// TIA Portal V19 program export: 0 tag tables, 0 data types, 49 data blocks, 112 code blocks (in call order from the OBs), 34 instance data blocks

DATA_BLOCK "Analogwerte"   // DB1110
{ S7_Optimized_Access := 'TRUE' }
// stored: AutoNumber false, MemoryReserve 100
   VAR RETAIN
      "LF_CM01.BN01" : Struct   // Leitfähigkeit Bypass Filterpumpe
         MB_min : Real := 0.0;
         MB_max : Real := 2000.0;   // mS
         UG_Alarm : Real := -0.5;
         OG_Alarm : Real := 2200.0;
         GF : Real := 0.5;
         Drahtbruch : Bool := FALSE;
         ungueltig : Bool := FALSE;
      END_STRUCT;
      "LF_CM01.BN02" : Struct   // Leitfähigkeit Düsen Umwälzung
         MB_min : Real := 0.0;
         MB_max : Real := 2000.0;   // mS
         UG_Alarm : Real := -0.5;
         OG_Alarm : Real := 2200.0;
         GF : Real := 0.5;
         Drahtbruch : Bool := FALSE;
         ungueltig : Bool := FALSE;
      END_STRUCT;
      "LF_CM02.BN03" : Struct   // Leitfähigkeit Bypass Filterpumpe
         MB_min : Real := 0.0;
         MB_max : Real := 2000.0;   // mS
         UG_Alarm : Real := -0.5;
         OG_Alarm : Real := 2200.0;
         GF : Real := 0.5;
         Drahtbruch : Bool := FALSE;
         ungueltig : Bool := FALSE;
      END_STRUCT;
      "LF_CM02.BN04" : Struct   // Leitfähigkeit Düsen Umwälzung
         MB_min : Real := 0.0;
         MB_max : Real := 2000.0;   // mS
         UG_Alarm : Real := -0.5;
         OG_Alarm : Real := 2200.0;
         GF : Real := 0.5;
         Drahtbruch : Bool := FALSE;
         ungueltig : Bool := FALSE;
      END_STRUCT;
      "p_HQ01.BP01" : Struct   // Druck Beutelfiltergehäuse
         MB_min : Real := 0.0;
         MB_max : Real := 4.0;   // bar
         UG_Alarm : Real := -0.5;
         OG_Alarm : Real := 4.5;
         GF : Real := 0.5;
         Drahtbruch : Bool := FALSE;
         ungueltig : Bool := FALSE;
      END_STRUCT;
      "p_HQ02.BP02" : Struct   // Druck Beutelfiltergehäuse
         MB_min : Real := 0.0;
         MB_max : Real := 4.0;   // bar
         UG_Alarm : Real := -0.5;
         OG_Alarm : Real := 4.5;
         GF : Real := 0.5;
         Drahtbruch : Bool := FALSE;
         ungueltig : Bool := FALSE;
      END_STRUCT;
      "p_CM01.BP03" : Struct   // Druck Filterpumpe
         MB_min : Real := 0.0;
         MB_max : Real := 4.0;   // bar
         UG_Alarm : Real := -0.5;
         OG_Alarm : Real := 4.5;
         GF : Real := 0.5;
         Drahtbruch : Bool := FALSE;
         ungueltig : Bool := FALSE;
      END_STRUCT;
      "p_CM01.BP04" : Struct   // Druck Umwälzpumpe
         MB_min : Real := 0.0;
         MB_max : Real := 4.0;   // bar
         UG_Alarm : Real := -0.5;
         OG_Alarm : Real := 4.5;
         GF : Real := 0.5;
         Drahtbruch : Bool := FALSE;
         ungueltig : Bool := FALSE;
      END_STRUCT;
      "p_CM03.BP05" : Struct   // Druck Umwäzpumpe
         MB_min : Real := 0.0;
         MB_max : Real := 4.0;   // bar
         UG_Alarm : Real := -0.5;
         OG_Alarm : Real := 4.5;
         GF : Real := 0.5;
         Drahtbruch : Bool := FALSE;
         ungueltig : Bool := FALSE;
      END_STRUCT;
      "p_CM02.BP06" : Struct   // Druck Filterpumpe
         MB_min : Real := 0.0;
         MB_max : Real := 4.0;   // bar
         UG_Alarm : Real := -0.5;
         OG_Alarm : Real := 4.5;
         GF : Real := 0.5;
         Drahtbruch : Bool := FALSE;
         ungueltig : Bool := FALSE;
      END_STRUCT;
      "p_CM02.BP07" : Struct   // Druck Umwälzpumpe
         MB_min : Real := 0.0;
         MB_max : Real := 4.0;   // bar
         UG_Alarm : Real := -0.5;
         OG_Alarm : Real := 4.5;
         GF : Real := 0.5;
         Drahtbruch : Bool := FALSE;
         ungueltig : Bool := FALSE;
      END_STRUCT;
      "p_CM04.BP08" : Struct   // Druck Umwäzpumpe
         MB_min : Real := 0.0;
         MB_max : Real := 4.0;   // bar
         UG_Alarm : Real := -0.5;
         OG_Alarm : Real := 4.5;
         GF : Real := 0.5;
         Drahtbruch : Bool := FALSE;
         ungueltig : Bool := FALSE;
      END_STRUCT;
      "p_CM05.BP09" : Struct   // Druck Pumpe Entleerung Sammeltank
         MB_min : Real := 0.0;
         MB_max : Real := 4.0;   // bar
         UG_Alarm : Real := -0.5;
         OG_Alarm : Real := 4.5;
         GF : Real := 0.5;
         Drahtbruch : Bool := FALSE;
         ungueltig : Bool := FALSE;
      END_STRUCT;
      "Dfl_GP01.BF01" : Struct   // Durchfluss Versorgung Frischsäure
         MB_min : Real := 0.0;
         MB_max : Real := 2000.0;   // ml/s
         UG_Alarm : Real := -0.5;
         OG_Alarm : Real := 2200.0;
         GF : Real := 0.5;
         Drahtbruch : Bool := FALSE;
         ungueltig : Bool := FALSE;
      END_STRUCT;
      "Dfl_GP02.BF02" : Struct   // Durchfluss Entsorgung Altsäure
         MB_min : Real := 0.0;
         MB_max : Real := 2000.0;   // ml/s
         UG_Alarm : Real := -0.5;
         OG_Alarm : Real := 2200.0;
         GF : Real := 0.5;
         Drahtbruch : Bool := FALSE;
         ungueltig : Bool := FALSE;
      END_STRUCT;
      "Niv_GP01.BL30" : Struct   // Füllstand Versorgung Frischsäure
         MB_min : Real := 0.0;
         MB_max : Real := 100.0;   // %
         UG_Alarm : Real := -0.5;
         OG_Alarm : Real := 110.0;
         GF : Real := 0.5;
         Drahtbruch : Bool := FALSE;
         ungueltig : Bool := FALSE;
      END_STRUCT;
      "Niv_GP02.BL31" : Struct   // Füllstand Entsorgung Altsäure
         MB_min : Real := 0.0;
         MB_max : Real := 100.0;   // %
         UG_Alarm : Real := -0.5;
         OG_Alarm : Real := 110.0;
         GF : Real := 0.5;
         Drahtbruch : Bool := FALSE;
         ungueltig : Bool := FALSE;
      END_STRUCT;
      pH_WR01 : Struct   // pH-Wert Be-/Entladen
         MB_min : Real := 0.0;
         MB_max : Real := 100.0;   // %
         UG_Alarm : Real := -0.5;
         OG_Alarm : Real := 110.0;
         GF : Real := 0.5;
         Drahtbruch : Bool := FALSE;
         ungueltig : Bool := FALSE;
      END_STRUCT;
      WZ_1_1 : Struct   // Wägezelle WR04.BW01
         MB_min : Real := 0.0;
         MB_max : Real := 100.0;   // %
         UG_Alarm : Real := -0.5;
         OG_Alarm : Real := 110.0;
         GF : Real := 0.5;
         Drahtbruch : Bool := FALSE;
         ungueltig : Bool := FALSE;
      END_STRUCT;
      WZ_1_2 : Struct   // Wägezelle WR04.BW02
         MB_min : Real := 0.0;
         MB_max : Real := 100.0;   // %
         UG_Alarm : Real := -0.5;
         OG_Alarm : Real := 110.0;
         GF : Real := 0.5;
         Drahtbruch : Bool := FALSE;
         ungueltig : Bool := FALSE;
      END_STRUCT;
      WZ_1_3 : Struct   // Wägezelle WR04.BW03
         MB_min : Real := 0.0;
         MB_max : Real := 100.0;   // %
         UG_Alarm : Real := -0.5;
         OG_Alarm : Real := 110.0;
         GF : Real := 0.5;
         Drahtbruch : Bool := FALSE;
         ungueltig : Bool := FALSE;
      END_STRUCT;
      WZ_1_4 : Struct   // Wägezelle WR04.BW04
         MB_min : Real := 0.0;
         MB_max : Real := 100.0;   // %
         UG_Alarm : Real := -0.5;
         OG_Alarm : Real := 110.0;
         GF : Real := 0.5;
         Drahtbruch : Bool := FALSE;
         ungueltig : Bool := FALSE;
      END_STRUCT;
      WZ_2_1 : Struct   // Wägezelle WR05.BW01
         MB_min : Real := 0.0;
         MB_max : Real := 100.0;   // %
         UG_Alarm : Real := -0.5;
         OG_Alarm : Real := 110.0;
         GF : Real := 0.5;
         Drahtbruch : Bool := FALSE;
         ungueltig : Bool := FALSE;
      END_STRUCT;
      WZ_2_2 : Struct   // Wägezelle WR05.BW01
         MB_min : Real := 0.0;
         MB_max : Real := 100.0;   // %
         UG_Alarm : Real := -0.5;
         OG_Alarm : Real := 110.0;
         GF : Real := 0.5;
         Drahtbruch : Bool := FALSE;
         ungueltig : Bool := FALSE;
      END_STRUCT;
      WZ_2_3 : Struct   // Wägezelle WR05.BW01
         MB_min : Real := 0.0;
         MB_max : Real := 100.0;   // %
         UG_Alarm : Real := -0.5;
         OG_Alarm : Real := 110.0;
         GF : Real := 0.5;
         Drahtbruch : Bool := FALSE;
         ungueltig : Bool := FALSE;
      END_STRUCT;
      WZ_2_4 : Struct   // Wägezelle WR05.BW01
         MB_min : Real := 0.0;
         MB_max : Real := 100.0;   // %
         UG_Alarm : Real := -0.5;
         OG_Alarm : Real := 110.0;
         GF : Real := 0.5;
         Drahtbruch : Bool := FALSE;
         ungueltig : Bool := FALSE;
      END_STRUCT;
      Last_1 : Struct   // Novamat WR04.BW34
         MB_min : Real := 0.0;
         MB_max : Real := 100.0;   // %
         UG_Alarm : Real := -0.5;
         OG_Alarm : Real := 110.0;
         GF : Real := 0.5;
         Drahtbruch : Bool := FALSE;
         ungueltig : Bool := FALSE;
      END_STRUCT;
      Last_2 : Struct   // Novamat WR05.BW43
         MB_min : Real := 0.0;
         MB_max : Real := 100.0;   // %
         UG_Alarm : Real := -0.5;
         OG_Alarm : Real := 110.0;
         GF : Real := 0.5;
         Drahtbruch : Bool := FALSE;
         ungueltig : Bool := FALSE;
      END_STRUCT;
   END_VAR
BEGIN
END_DATA_BLOCK

DATA_BLOCK "DB_ANLAGE"   // DB1
{ S7_Optimized_Access := 'FALSE' }
AUTHOR : MS
// stored: AutoNumber false
   VAR RETAIN
      BA : Struct   // Betriebsarten
         Not_Aus : Bool := FALSE;   // Not-Aus ist betätigt
         free0 : Bool := FALSE;   // sonst Anlage vom PC bedienen, nur bei BA-Schalter auf Auto
         free1 : Bool := FALSE;   // sonst Automatikbetrieb ist nicht freigegeben
         Tippbetrieb : Bool := FALSE;   // Tippbetrieb
         Handbetrieb : Bool := FALSE;   // Handbetrieb
         Automat_ein : Bool := FALSE;   // Automatikbetrieb möglich
         Automat_aus : Bool := FALSE;   // Automatikbetrieb nicht möglich
         Anlauf_Auto : Bool := FALSE;   // Anlauf Automatik für Scanvorgang WT-Positionen auf letzte Automatikposition
         Einfahr_Stop : Bool := FALSE;   // Stoppt die Einfahrt von WT in die Anlage(Feierabendprogramm)
         Mess_on : Bool := FALSE;   // Einmessung aktiv
         Taktwechsel : Bool := FALSE;   // Taktwechsel durchführen
         SIM_HISPEED : Bool := FALSE;   // * Simulation erfolgt mit doppelter Geschwindigkeit
         Simulation : Bool := FALSE;   // * Simulation eingeschaltet
         COM_RST : Bool := TRUE;   // Complete Restart
         FP_Automat_ein : Bool := FALSE;   // Flankenmerker positive Flanke Taste Automat ein
         newConfig : Bool := FALSE;   // neue Konfiguration (Daten neu verteilen)
      END_STRUCT;
      config : Struct   // Anlagenkonfiguration
         ANZ_FW : Int := 1;   // * Anzahl der Transportwagen in der Anlage
         ANZ_QT : Int := 0;   // * Anzahl der Quertransporte in der Anlage
         ANZ_Reihen : Int := 1;   // * Anzahl der Reihen in der Anlage
         ANZ_Pos : Int := 30;   // * Anzahl der Positionen
         ANZ_WT : Int := 12;   // * Anzahl der vorhandenen WT-Datenbausteine
         ANZ_POS_per_Cyc : Int := 6;   // * Anzahl der bearbeiteten Positionen pro Zyklus
         maxWT_loop : Int := 5;   // * im freien System Anzahl der Befehle der größten Technologieschleife
         Anz_Opt_Pos : Int := 0;   // * Anzahl der in die Optimierungsrechnung eingehenden Positionen
         Anz_GR : Int := 0;   // * Anzahl der Gleichrichter
         Anz_TR : Int := 0;   // * Anzahl der Temperaturregler
         Anz_DZ : Int := 2;   // * Anzahl der Dosierzähler
         Anz_DP : Int := 8;   // * Anzahl Dosierpumpen
         AnaEventInt : Int := 600;   // * Analogevent Intervall
         Taktzeit_typ : Int := 480;   // * typische Taktzeit für Expoberechnung in getakteten Positionen
         Transzeit_typ : Int := 60;   // * typische Zeit für einen Austauschvorgang
         Reihen_Cnfg : Struct
            EndePos_R1 : Int := 30;   // * Reihendefinition, letzte Position in Reihe 1 (immer niedriger als EndePos_R2)
            EndePos_R2 : Int := 0;   // * Reihendefinition, letzte Position in Reihe 2 (immer niedriger als EndePos_R3)
            EndePos_R3 : Int := 0;   // * Reihendefinition, letzte Position in Reihe 3 (immer niedriger als EndePos_R4)
            EndePos_R4 : Int := 0;   // * Reihendefinition, letzte Position in Reihe 4 (immer niedriger als EndePos_R5)
            EndePos_R5 : Int := 0;   // * Reihendefinition, letzte Position in Reihe 5
         END_STRUCT;
         akt_FW : Int := 0;
         Old_Hour_Event : Int := 0;
         PC_exist : Bool := 0;   // * PC-Daten schreiben (es existiert ein EventAbnehmer [FC7])
         Diag_exist : Bool := 0;   // * Diagrammdaten schreiben (Diagrammdaten werden am PC aufgezeichnet)
         Anl_getaktet : Bool := TRUE;   // * 0=Anlage fährt Auftragsorientiert 1=Anlage wird mit Ketten gesteuert
         HW_exist : Bool := TRUE;   // * Höhenwechsel in der Anlage vorhanden
         Pos_absolut : Bool := TRUE;   // * Positionsbestimmung absolut für OB100-Init-Pos (wirkt nicht mehr am FW)
         Opti_exist : Bool := FALSE;   // * Optimierung vorhanden
         AL_Einfahrt : Bool := FALSE;   // Ware aufgeben!!
         Al_Ausfahrt : Bool := FALSE;   // Beladestand räumen!!
         Weg_Zeit_aus : Bool := FALSE;   // * Weg-Zeit-Events nicht schreiben
         EntmFromOpt : Bool := FALSE;   // * Entmetallisierungs-WT werden von der Optimierung berechnet
         M_Q_Hupe : Bool := TRUE;
         HW_Auto_search : Bool := FALSE;   // * FW sucht automatisch nach einer möglichen Höhenwechselposition
         FP_Taste_Reset : Bool := FALSE;
         Time_from_PC : Bool := 0;   // * Zeit wird vom PC gestellt (keine autom. Sommerzeit)
         FP_Stop_Taktende : Bool := FALSE;   // Flankenmerker Stop bei Taktende erreicht
         Temp_MW_aktiv : Bool := 0;   // * Event mittlere Temperatur (Event 18) aktiv
         FP_Einrichten : Bool := FALSE;
         FP_Hand : Bool := TRUE;
         FP_Automatik : Bool := FALSE;
         FP_In_Quitt : Bool := FALSE;   // Flankenmerker Fehlerquittung
         Hub_absolut : Bool := FALSE;   // Hubsesorik Absolutgeber
         Battf : Bool := FALSE;   // Batteriefehler OB81 (Durch Hardwareschalter an SPS "BATT_INDIC") quittierbar
         RESET_STATUS : Bool := FALSE;   // Wiederanlaufmerker nach Reset
         WT_Typ_Afg : Bool := FALSE;   // * WT-Typ wird bei Aufgabe vergeben
         TypChckDetail : Bool := TRUE;   // * WT-Typ wird ohne Maske B#16#F0 geprüft
         QT_Trocken_chk : Bool := FALSE;   // * einschalten, wenn Prüfung auf bit "immer schnell"
         FB9_Takt : Bool := FALSE;   // * FB9 aufrufen obwohl Anlage getaktet
         Use_FB_Ana : Bool := 0;   // * 1=FB110 verwenden 0=klassische Analogwerterfassung FC110
         Check_Profibus : Bool := TRUE;   // * Profibusteilnehmer überwachen! OB86,OB100,DB203,FC203
         NormalB : Bool := FALSE;   // 0: 151 / 161 1: nur 151
         res6 : Bool := FALSE;
         ReqUmsTakt : Bool := FALSE;   // Anforderung Umschaltung auf getaktet
      END_STRUCT;
      IN : Struct   // Hardwareeingänge Anlage
         S_Not_Aus : Bool := FALSE;   // Not-Aus ok
         S_St_Spng : Bool := TRUE;   // Steuerspannung ein
         Quitt_Err : Bool := FALSE;   // Fehlerquittung
         Quitt_Hupe : Bool := FALSE;   // Hupenquittierung
         Reset : Bool := FALSE;   // Reset Anlagenschalter
         Reparatur : Bool := FALSE;   // Reparaturbetrieb
         Lamp_Test : Bool := FALSE;   // Lampentest
         BA_Tipp : Bool := FALSE;   // BA Umschalter Tipp
         BA_Hand : Bool := TRUE;   // BA Umschalter Hand
         BA_Auto : Bool := FALSE;   // BA Umschalter Auto
         Stop_Anlage : Bool := FALSE;   // Anlage hält am Takt- bzw. Schichtende an
         Automat_aus : Bool := FALSE;   // Taste Automatikbetrieb verbieten
         Automat_ein : Bool := FALSE;   // Taste Automatikbetrieb erlauben
         Quit_Err_Galva : Bool := FALSE;   // Fehlerquittung per Galva
         res4 : Bool := FALSE;
         UT_Req : Bool := FALSE;   // Anforderung Umlufttrockner
         ReqEventTakt : Bool := FALSE;   // Anforderung EventTakt
         GR_ok : Bool := FALSE;   // Rückmeldung Event erfolgt
         TR_ok : Bool := FALSE;   // Rückmeldung Event erfolgt
         pH_LF_ok : Bool := TRUE;   // Rückmeldung Event erfolgt
         DP_ok : Bool := FALSE;   // Rückmeldung Event erfolgt
         res11 : Bool := FALSE;
         res12 : Bool := FALSE;
         res13 : Bool := FALSE;
         PC_offline : Bool := FALSE;   // PC-Komunikation ist unterbrochen
         AMS_Restart : Bool := FALSE;   // alle anstehenden Fehler neu senden
         Watch_Profibus : Bool := FALSE;   // Profibusüberwachung eingeschaltet
         res17 : Bool := FALSE;
         res18 : Bool := FALSE;
         res19 : Bool := FALSE;
         res20 : Bool := FALSE;
         AMS_Reset : Bool := FALSE;   // AMS-Reset durchführen (Resetknopf während nicht Tipp)
      END_STRUCT;
      OUT : Struct   // Hardwareausgänge Anlage
         Stoerung_Opt : Bool := FALSE;
         Stoerung_Aku : Bool := FALSE;
         MD_Auto : Bool := FALSE;
         Fehler_Quitt : Bool := FALSE;
         res1 : Bool := FALSE;
         res2 : Bool := FALSE;
         res3 : Bool := FALSE;
         FW_QT_Auto : Bool := FALSE;   // mind. ein FW/QT hat seinen Automatikbefehl noch nicht beendet
         TW_abgelehnt : Bool := FALSE;   // Taktwechsel wurde abgelehnt (durch Fehlerquittung löschen)
         WT_in_Anlage : Bool := FALSE;
         res7 : Bool := FALSE;
         res8 : Bool := FALSE;
         res9 : Bool := FALSE;
         res10 : Bool := FALSE;
         res11 : Bool := FALSE;
         res12 : Bool := FALSE;
         res13 : Bool := FALSE;
         res14 : Bool := FALSE;
         res15 : Bool := FALSE;
         res16 : Bool := FALSE;
         res17 : Bool := FALSE;
         res18 : Bool := FALSE;
         res19 : Bool := FALSE;
         res20 : Bool := FALSE;
         AnzUT_Req : Byte := 16#00;   // Anzahl der UT Anforderungen
      END_STRUCT;
      config2 : Struct
         Anzahl_HW : Int := 1;   // * Anzahl Höhenwechsel (Definition im DB53)
         Woscha_DB_1 : Int := 8;   // Datenbaustein für Wochenschaltuhr 1
         Woscha_DB_2 : Int := 0;   // Datenbaustein für Wochenschaltuhr 2
         Woscha_DB_3 : Int := 0;   // Datenbaustein für Wochenschaltuhr 3
         Woscha_DB_4 : Int := 0;   // Datenbaustein für Wochenschaltuhr 4
         resW4 : Int := 0;
         Anlagentakte : Int := 3;   // Anzahl Takte, welche WT durch die Anlage läuft
         resW6 : Int := 0;
         resW7 : Int := 0;
         resW8 : Int := 0;
         resW9 : Int := 0;
         resW10 : Int := 0;
         resW11 : Int := 0;
         resW12 : Int := 0;
         resW13 : Int := 0;
         resW14 : Int := 0;
         resW15 : Int := 0;
         resW16 : Int := 0;
         resW17 : Int := 0;
         resW18 : Int := 0;
         resW19 : Int := 0;
      END_STRUCT;
      FW1 : Struct
         FW_min : Int := 1;   // * FW Bereich min
         FW_max : Int := 30;   // * FW Bereich max
         RefPos : Int := 0;   // * Referenzposition (bei Absolutpositionierung 0)
         T_Nr : Int := 10;   // * Timer1
         resW : Int := 0;
      END_STRUCT;
      FW2 : Struct
         FW_min : Int := 0;   // * FW Bereich min
         FW_max : Int := 0;   // * FW Bereich max
         RefPos : Int := 0;   // * Referenzposition (bei Absolutpositionierung 0)
         T_Nr : Int := 0;   // * Timer1
         resW : Int := 0;
      END_STRUCT;
      FW3 : Struct
         FW_min : Int := 0;   // * FW Bereich min
         FW_max : Int := 0;   // * FW Bereich max
         RefPos : Int := 0;   // * Referenzposition (bei Absolutpositionierung 0)
         T_Nr : Int := 0;   // * Timer1
         resW : Int := 0;
      END_STRUCT;
      FW4 : Struct
         FW_min : Int := 0;   // * FW Bereich min
         FW_max : Int := 0;   // * FW Bereich max
         RefPos : Int := 0;   // * Referenzposition (bei Absolutpositionierung 0)
         T_Nr : Int := 0;   // * Timer1
         resW : Int := 0;
      END_STRUCT;
      FW5 : Struct
         FW_min : Int := 0;   // * FW Bereich min
         FW_max : Int := 0;   // * FW Bereich max
         RefPos : Int := 0;   // * Referenzposition (bei Absolutpositionierung 0)
         T_Nr : Int := 0;   // * Timer1
         resW : Int := 0;
      END_STRUCT;
      FW6 : Struct
         FW_min : Int := 0;   // * FW Bereich min
         FW_max : Int := 0;   // * FW Bereich max
         RefPos : Int := 0;   // * Referenzposition (bei Absolutpositionierung 0)
         T_Nr : Int := 0;   // * Timer1
         resW : Int := 0;
      END_STRUCT;
      FW7 : Struct
         FW_min : Int := 0;   // * FW Bereich min
         FW_max : Int := 0;   // * FW Bereich max
         RefPos : Int := 0;   // * Referenzposition (bei Absolutpositionierung 0)
         T_Nr : Int := 0;   // * Timer1
         resW : Int := 0;
      END_STRUCT;
      FW8 : Struct
         FW_min : Int := 0;   // * FW Bereich min
         FW_max : Int := 0;   // * FW Bereich max
         RefPos : Int := 0;   // * Referenzposition (bei Absolutpositionierung 0)
         T_Nr : Int := 0;   // * Timer1
         resW : Int := 0;
      END_STRUCT;
      FW9 : Struct
         FW_min : Int := 0;   // * FW Bereich min
         FW_max : Int := 0;   // * FW Bereich max
         RefPos : Int := 0;   // * Referenzposition (bei Absolutpositionierung 0)
         T_Nr : Int := 0;   // * Timer1
         resW : Int := 0;
      END_STRUCT;
      FW10 : Struct
         FW_min : Int := 0;   // * FW Bereich min
         FW_max : Int := 0;   // * FW Bereich max
         RefPos : Int := 0;   // * Referenzposition (bei Absolutpositionierung 0)
         T_Nr : Int := 0;   // * Timer1
         resW : Int := 0;
      END_STRUCT;
      FW11 : Struct
         FW_min : Int := 0;   // * FW Bereich min
         FW_max : Int := 0;   // * FW Bereich max
         RefPos : Int := 0;   // * Referenzposition (bei Absolutpositionierung 0)
         T_Nr : Int := 0;   // * Timer1
         resW : Int := 0;
      END_STRUCT;
      FW12 : Struct
         FW_min : Int := 0;   // * FW Bereich min
         FW_max : Int := 0;   // * FW Bereich max
         RefPos : Int := 0;   // * Referenzposition (bei Absolutpositionierung 0)
         T_Nr : Int := 0;   // * Timer1
         resW : Int := 0;
      END_STRUCT;
      FW13 : Struct
         FW_min : Int := 0;   // * FW Bereich min
         FW_max : Int := 0;   // * FW Bereich max
         RefPos : Int := 0;   // * Referenzposition (bei Absolutpositionierung 0)
         T_Nr : Int := 0;   // * Timer1
         resW : Int := 0;
      END_STRUCT;
      FW14 : Struct
         FW_min : Int := 0;   // * FW Bereich min
         FW_max : Int := 0;   // * FW Bereich max
         RefPos : Int := 0;   // * Referenzposition (bei Absolutpositionierung 0)
         T_Nr : Int := 0;   // * Timer1
         resW : Int := 0;
      END_STRUCT;
      FW15 : Struct
         FW_min : Int := 0;   // * FW Bereich min
         FW_max : Int := 0;   // * FW Bereich max
         RefPos : Int := 0;   // * Referenzposition (bei Absolutpositionierung 0)
         T_Nr : Int := 0;   // * Timer1
         resW : Int := 0;
      END_STRUCT;
      QT1 : Struct
         PosR1 : Byte := 16#00;   // * QT-Reihe1: Positionsnummer der ersten QT-Pos (bei Rückwärtsfahrt letzte Pos)
         PosR2 : Byte := 16#00;   // * QT-Reihe2: Positionsnummer der zweiten QT-Pos
         PosR3 : Byte := 16#00;   // * QT-Reihe3: Positionsnummer der dritten QT-Pos
         PosR4 : Byte := 16#00;   // * QT-Reihe4: Positionsnummer der vierten QT-Pos
         PosR5 : Byte := 16#00;   // * QT-Reihe5: Positionsnummer der fünften QT-Pos
         RefReihe : Byte := 16#00;   // * Referenzreihe nur angeben wenn mitfahrende Sensoren!!
         T_Nr : Int := 0;   // * Timer1
         Ketten_DB : Int := 0;   // * Eintrag == 0 --> QT besitzt keine Kette
      END_STRUCT;
      QT2 : Struct
         PosR1 : Byte := 16#00;   // * QT-Reihe1: Positionsnummer der ersten QT-Pos (bei Rückwärtsfahrt letzte Pos)
         PosR2 : Byte := 16#00;   // * QT-Reihe2: Positionsnummer der zweiten QT-Pos
         PosR3 : Byte := 16#00;   // * QT-Reihe3: Positionsnummer der dritten QT-Pos
         PosR4 : Byte := 16#00;   // * QT-Reihe4: Positionsnummer der vierten QT-Pos
         PosR5 : Byte := 16#00;   // * QT-Reihe5: Positionsnummer der fünften QT-Pos
         RefReihe : Byte := 16#00;   // * Referenzreihe nur angeben wenn mitfahrende Sensoren!!
         T_Nr : Int := 0;   // * Timer1
         Ketten_DB : Int := 0;   // * Eintrag == 0 --> QT besitzt keine Kette
      END_STRUCT;
      QT3 : Struct
         PosR1 : Byte := 16#00;   // * QT-Reihe1: Positionsnummer der ersten QT-Pos (bei Rückwärtsfahrt letzte Pos)
         PosR2 : Byte := 16#00;   // * QT-Reihe2: Positionsnummer der zweiten QT-Pos
         PosR3 : Byte := 16#00;   // * QT-Reihe3: Positionsnummer der dritten QT-Pos
         PosR4 : Byte := 16#00;   // * QT-Reihe4: Positionsnummer der vierten QT-Pos
         PosR5 : Byte := 16#00;   // * QT-Reihe5: Positionsnummer der fünften QT-Pos
         RefReihe : Byte := 16#00;   // * Referenzreihe nur angeben wenn mitfahrende Sensoren!!
         T_Nr : Int := 0;   // * Timer1
         Ketten_DB : Int := 0;   // * Eintrag == 0 --> QT besitzt keine Kette
      END_STRUCT;
      QT4 : Struct
         PosR1 : Byte := 16#00;   // * QT-Reihe1: Positionsnummer der ersten QT-Pos (bei Rückwärtsfahrt letzte Pos)
         PosR2 : Byte := 16#00;   // * QT-Reihe2: Positionsnummer der zweiten QT-Pos
         PosR3 : Byte := 16#00;   // * QT-Reihe3: Positionsnummer der dritten QT-Pos
         PosR4 : Byte := 16#00;   // * QT-Reihe4: Positionsnummer der vierten QT-Pos
         PosR5 : Byte := 16#00;   // * QT-Reihe5: Positionsnummer der fünften QT-Pos
         RefReihe : Byte := 16#00;   // * Referenzreihe nur angeben wenn mitfahrende Sensoren!!
         T_Nr : Int := 0;   // * Timer1
         Ketten_DB : Int := 0;   // * Eintrag == 0 --> QT besitzt keine Kette
      END_STRUCT;
      QT5 : Struct
         PosR1 : Byte := 16#00;   // * QT-Reihe1: Positionsnummer der ersten QT-Pos (bei Rückwärtsfahrt letzte Pos)
         PosR2 : Byte := 16#00;   // * QT-Reihe2: Positionsnummer der zweiten QT-Pos
         PosR3 : Byte := 16#00;   // * QT-Reihe3: Positionsnummer der dritten QT-Pos
         PosR4 : Byte := 16#00;   // * QT-Reihe4: Positionsnummer der vierten QT-Pos
         PosR5 : Byte := 16#00;   // * QT-Reihe5: Positionsnummer der fünften QT-Pos
         RefReihe : Byte := 16#00;   // * Referenzreihe nur angeben wenn mitfahrende Sensoren!!
         T_Nr : Int := 0;   // * Timer1
         Ketten_DB : Int := 0;   // * Eintrag == 0 --> QT besitzt keine Kette
      END_STRUCT;
   END_VAR
BEGIN
END_DATA_BLOCK

DATA_BLOCK "DB_Alarme"   // DB1201
{ S7_Optimized_Access := 'TRUE' }
// stored: AutoNumber false, MemoryReserve 100
   VAR RETAIN
      MLD : Array[0.."Anzahl_Alarm_Woerter"] of Word;
      AM_MLD : Array[0.."Anzahl_Alarm_Woerter"] of Word;
      Para_Mld : Array[0.."Anzahl_Alarm_Woerter"] of "Alarm_Parameter_Wort";   // Struct = Meldewort, Array = ParaByte für MeldeBit (siehe FC5)
      WrnM : Array[0..1] of Word;
      Edit : Struct
         Edit_Meld : Int := 1;   // aktuell zu editierende Meldung
         Edit_Meld_old : Int;
         Edit_Meldewort : Int;   // betroffenes Meldewort
         Edit_Meldebit : Int;   // betroffenes Meldebit
         AM_Edit : Bool;
         Uebernehmen : Bool;   // Änderungen Übernehmen
         Uebernommen : Bool;   // Änderungen für ausgewählte Meldung übernommen
         Verwerfen : Bool;   // Änderungen verwerfen
         Editiert : Bool;   // Alarm wurde geändert
         Par : "Alarm_Parameter";
      END_STRUCT;
      auto_aus : Bool;
      stop_request : Bool;
      Sammelbit_St : Bool;
      Sammelbit_Wrn : Bool;
      M_Q_Hupe_Rot : Bool;
      M_Q_Hupe_Gelb : Bool;
      M_Q_Hupe_Blau : Bool;
      Hupe_Dauer_Rot : Bool;
      Hupe_Dauer_Gelb : Bool;
      Hupe_Dauer_Blau : Bool;
      IN_Quitt_Hupe : Bool;
      AM_T_Hupe : Bool;
      La_Quit_Err : Bool;   // Lampe Fehlerquittung
      Lampe_Rot : Bool;
      Lampe_Gelb : Bool;
      Lampe_Blau : Bool;
      Zeit_Auto_Quitt_Hupe_Rot : Time_Of_Day := TOD#00:00:05;
      Zeit_Auto_Quitt_Hupe_Gelb : Time_Of_Day := TOD#00:00:05;
      Zeit_Auto_Quitt_Hupe_Blau : Time_Of_Day := TOD#00:00:05;
      Timer_Hupe_Rot : TON_TIME;
      Timer_Hupe_Gelb : TON_TIME;
      Timer_Hupe_Blau : TON_TIME;
   END_VAR
BEGIN
END_DATA_BLOCK

DATA_BLOCK "DB_DP_Error"   // DB203
{ S7_Optimized_Access := 'FALSE' }
// stored: AutoNumber false
   VAR
      DP_Slave : Array[0..1023] of Byte;   // 0..n.v.,nicht projektiert,1..vorhanden,ok,2..vorhanden,nok,3..projektiert,n.v.
      Altwert : Array[0..1023] of Byte;   // 0..n.v.,nicht projektiert,1..vorhanden,ok,2..vorhanden,nok,3..projektiert,n.v.
      HiAdr : Int;   // höchste Teilnehmeradresse
      Init : Bool;   // Anlaufzyklus oder AMS-Reset --> Initialisierung
      Hupe_enable : Bool;   // * Hupe bei Alarm einschalten?
      Sammelstoerung : Bool;   // Störung/Ausfall
      Sammelwarnung : Bool;   // Warnung/Fehler einer Baugruppe
      res1 : Bool;
      res2 : Bool;
      res3 : Bool;
      res4 : Bool;
   END_VAR
BEGIN
END_DATA_BLOCK

DATA_BLOCK "DB_Daten_Heraeus"   // DB1111
{ S7_Optimized_Access := 'FALSE' }
// stored: AutoNumber false
   VAR RETAIN
      "Leitwert_CM01.BN01" : Real;   // Leitfähigkeit Bypass Filterpumpe
      "Leitwert_CM01.BN02" : Real;   // Leitfähigkeit Düsen Umwälzung
      "Leitwert_CM02.BN03" : Real;   // Leitfähigkeit Bypass Filterpumpe
      "Leitwert_CM02.BN04" : Real;   // Leitfähigkeit Düsen Umwälzung
      "p_HQ01.BP01" : Real;   // Druck Beutelfiltergehäuse
      "p_HQ02.BP02" : Real;   // Druck Beutelfiltergehäuse
      "p_CM01.BP03" : Real;   // Druck Filterpumpe
      "p_CM01.BP04" : Real;   // Druck Umwälzpumpe
      "p_CM03.BP05" : Real;   // Druck Umwäzpumpe
      "p_CM02.BP06" : Real;   // Druck Filterpumpe
      "p_CM02.BP07" : Real;   // Druck Umwälzpumpe
      "p_CM04.BP08" : Real;   // Druck Umwäzpumpe
      "p_CM05.BP09" : Real;   // Druck Pumpe Entleerung Sammeltank
   END_VAR
BEGIN
END_DATA_BLOCK

DATA_BLOCK "DB_Schaltuhr"   // DB1050
{ S7_Optimized_Access := 'TRUE' }
// stored: AutoNumber false, MemoryReserve 0
   VAR RETAIN
      Tag : Array[1..7] of Struct   // Tag 1: Sonntag
         AZ_Begin1 : DTL;   // Arbeitszeit Beginn
         AZ_Ende1 : DTL;   // Arbeitszeit Ende
         AZ_Begin2 : DTL;   // Arbeitszeit Beginn
         AZ_Ende2 : DTL;   // Arbeitszeit Ende
      END_STRUCT;
      Tag_aktiv : Array[1..7] of Struct   // Übertagung aktiv- oder deaktivieren
         AZ_Begin1_aktiv : Bool;   // =1, das Wort wird im SPS übertragen (nach Plausibilitätsprüfung)
         AZ_Ende1_aktiv : Bool;   // =1, das Wort wird im SPS übertragen (nach Plausibilitätsprüfung)
         AZ_Begin2_aktiv : Bool;   // =1, das Wort wird im SPS übertragen (nach Plausibilitätsprüfung)
         AZ_Ende2_aktiv : Bool;   // =1, das Wort wird im SPS übertragen (nach Plausibilitätsprüfung)
      END_STRUCT;
      Date_Time_Visu : DTL;   // fürs Uhrzeit stellen
      BA_Visu : Int;
      SPS_Zeit_holen : Bool;
      SPS_Zeit_Stellen : Bool;
      Taste_uebernehmen : Bool;   // Schaltuhreinträge Prüfen und Übernehmen
      Uebernommen : Bool;   // für sichtbarkeit von Button "Übernehmen in Visu"
      nichtOK : Bool;   // Meldung generieren wenn Eintrag niO
   END_VAR
BEGIN
END_DATA_BLOCK

DATA_BLOCK "DB_Temporaer"   // DB999
{ S7_Optimized_Access := 'TRUE' }
// stored: AutoNumber false, MemoryReserve 100
   VAR RETAIN
      Drucksensoren_deaktiviert : Bool;   // 20.01.22
   END_VAR
BEGIN
END_DATA_BLOCK

DATA_BLOCK "Drucktest"   // DB340
{ S7_Optimized_Access := 'FALSE' }
// stored: AutoNumber false
   VAR RETAIN
      akt_Index : Int := 0;
      Index_Panel : Int;
      Ergebnis : Array[0..100] of Struct
         "Name" : String[12];
         Zeit : DTL;
         ok : Bool;
         Fehler : Bool;
      END_STRUCT;
   END_VAR
BEGIN
END_DATA_BLOCK

DATA_BLOCK "MobilePanel"   // DB1071
{ S7_Optimized_Access := 'FALSE' }
// stored: AutoNumber false
   VAR
      Koordinierung : Word;
      Schluessel : Bool;
      Drucktaster_K2_LED : Int;
      Drucktaster_K2_Push : Bool;
   END_VAR
BEGIN
END_DATA_BLOCK

DATA_BLOCK "Panel"   // DB1070
{ S7_Optimized_Access := 'TRUE' }
// stored: AutoNumber false, MemoryReserve 100
   VAR RETAIN
      IW : Struct   // Analogwerte
         "LF_CM01.BN01" : Real;   // Leitfähigkeit Bypass Filterpumpe
         "LF_CM01.BN02" : Real;   // Leitfähigkeit Düsen Umwälzung
         "LF_CM02.BN03" : Real;   // Leitfähigkeit Bypass Filterpumpe
         "LF_CM02.BN04" : Real;   // Leitfähigkeit Düsen Umwälzung
         "p_HQ01.BP01" : Real;   // Druck Beutelfiltergehäuse
         "p_HQ02.BP02" : Real;   // Druck Beutelfiltergehäuse
         "p_CM01.BP03" : Real;   // Druck Filterpumpe
         "p_CM01.BP04" : Real;   // Druck Umwälzpumpe
         "p_CM03.BP05" : Real;   // Druck Umwäzpumpe
         "p_CM02.BP06" : Real;   // Druck Filterpumpe
         "p_CM02.BP07" : Real;   // Druck Umwälzpumpe
         "p_CM04.BP08" : Real;   // Druck Umwäzpumpe
         "p_CM05.BP09" : Real;   // Druck Pumpe Entleerung Sammeltank
         "Dfl_GP01.BF01" : Real;   // Durchfluss Versorgung Frischsäure
         "Dfl_GP02.BF02" : Real;   // Durchfluss Entsorgung Altsäure
         "Niv_GP01.BL30" : Real;   // Füllstand Versorgung Frischsäure
         "Niv_GP02.BL31" : Real;   // Füllstand Entsorgung Altsäure
         pH_BE : Real;   // SRM_Auf_BG-QM43
      END_STRUCT;
      Deckel : Struct   // Deckel Säurebecken
         CM01 : Struct
            Auto : Bool;
            Hand : Bool;
            Tipp : Bool;
            links_auf : Bool;
            links_zu : Bool;
            rechts_auf : Bool;
            rechts_zu : Bool;
            SRM_links_auf : Bool;
            SRM_links_zu : Bool;
            SRM_rechts_auf : Bool;
            SRM_rechts_zu : Bool;
            S_links_auf : Bool;   // CM01.BG01
            S_links_zu : Bool;   // CM01.BG02
            S_rechts_auf : Bool;   // CM01.BG03
            S_rechts_zu : Bool;   // CM01.BG04
            Ist_Pos_links : Int;   // 0% = auf; 100% = zu
            Ist_Pos_rechts : Int;   // 0% = auf; 100% = zu
         END_STRUCT;
         CM02 : Struct
            Auto : Bool;
            Hand : Bool;
            Tipp : Bool;
            links_auf : Bool;
            links_zu : Bool;
            rechts_auf : Bool;
            rechts_zu : Bool;
            SRM_links_auf : Bool;
            SRM_links_zu : Bool;
            SRM_rechts_auf : Bool;
            SRM_rechts_zu : Bool;
            S_links_auf : Bool;   // CM02.BG01
            S_links_zu : Bool;   // CM02.BG02
            S_rechts_auf : Bool;   // CM02.BG03
            S_rechts_zu : Bool;   // CM02.BG04
            Ist_Pos_links : Int;   // 0% = auf; 100% = zu
            Ist_Pos_rechts : Int;   // 0% = auf; 100% = zu
         END_STRUCT;
      END_STRUCT;
      RT : Struct   // Schnelllauftor
         K_Auto : Bool;   // Knauf Auto
         T_auf : Bool;   // Taste RT auf
         T_zu : Bool;   // Taste RT zu
         MSS_ok : Bool;   // Motorschutzschalter o.k.
         S_offen : Bool;   // Schnelllauftor offen
         S_geschlossen : Bool;   // Schnelllauftor geschlossen
         ok : Bool;   // Schnelllauftor o.k.
         Status : USInt;
      END_STRUCT;
      Ventilator : Struct   // FU[7]
         Ein : Bool;
         Auto : Bool;
         laeuft : Bool;
         betriebsbereit : Bool;
         Stoerung : Bool;
         Status : USInt;
         SW_Hand : Int;   // [%]
         SW_Auto_AZ : Int;   // [%]
         SW_Auto_aAZ : Int;   // [%]
         speed : Int;   // [%]
      END_STRUCT;
      CM01 : Struct   // HF-Becken 1
         Betrieb : Bool;
         Wartung : Bool;
         Niv_TGS : Bool;   // BL04
         Niv_Min : Bool;   // BL03
         Niv_max : Bool;   // BL02
         Niv_Uel : Bool;   // BL01
         NSP_Auto : Bool;
         GW_LF_FP : Bool;   // BN01
         GW_LF_UP : Bool;   // BN02
         GW_p_FP : Bool;   // BP03
         GW_p_UP : Bool;   // BP04
         Niv_Proz : USInt;
         Sollwert_LF : Real;   // Dosierung
         Dosierung_LF : Bool;   // 0 = WT, 1= LF
      END_STRUCT;
      CM02 : Struct   // HF-Becken 2
         Betrieb : Bool;
         Wartung : Bool;
         Niv_TGS : Bool;   // BL11
         Niv_Min : Bool;   // BL10
         Niv_max : Bool;   // BL09
         Niv_Uel : Bool;   // BL08
         NSP_Auto : Bool;
         GW_LF_FP : Bool;   // BN03
         GW_LF_UP : Bool;   // BN04
         GW_p_FP : Bool;   // BP06
         GW_p_UP : Bool;   // BP07
         Niv_Proz : USInt;
         Sollwert_LF : Real;   // Dosierung
         Dosierung_LF : Bool;   // 0 = WT, 1= LF
      END_STRUCT;
      CM03 : Struct   // Spülbecken 1
         Betrieb : Bool;
         Wartung : Bool;
         Niv_TGS : Bool;   // BL07
         Niv_Min : Bool;   // BL06
         GW_p_UP : Bool;   // BP05
         Niv_Proz : USInt;
         SPR_Auto : Bool;
         SPR_Start_Test : Bool;
         SPR_Stopp_Test : Bool;
         SPR_Zeit_Test : Int;
      END_STRUCT;
      CM04 : Struct   // Spülbecken 2
         Betrieb : Bool;
         Wartung : Bool;
         Niv_TGS : Bool;   // BL14
         Niv_Min : Bool;   // BL13
         GW_p_UP : Bool;   // BP08
         Niv_Proz : USInt;
         SPR_Auto : Bool;
         SPR_Start_Test : Bool;
         SPR_Stopp_Test : Bool;
         SPR_Zeit_Test : Int;
         NSP_Auto : Bool;
         NSP_Zeit : Int;   // pro Korb
         NSP_Start_Test : Bool;
         NSP_Stopp_Test : Bool;
         NSP_Zeit_Tes : Int;
      END_STRUCT;
      CM05 : Struct   // Abwassersammler
         Betrieb : Bool;
         Wartung : Bool;
         Niv_TGS : Bool;   // BL03
         Niv_Min : Bool;   // BL02
         Niv_max : Bool;   // BL01
         Niv_Uel : Bool;   // BL05
         AWA_Bereit : Bool;
         Frg_Abpumpen : Bool;
         GW_p_Pu : Bool;   // BP09
         Niv_Proz : USInt;
      END_STRUCT;
      HQ01 : Struct   // Filtereinheit
         Niv_Leckage : Bool;   // BL05
         GW_p_FG : Bool;   // BP01
         S_FG_zu : Bool;   // BG06
         S_Dkl_FG_li : Bool;   // BG07
         S_Dkl_FG_re : Bool;   // BG08
         Quitt_FW : Bool;
         Quitt_FW_erlaubt : Bool;
         WarnGr_FW : Real;
         Wechsel_FW : Real;
      END_STRUCT;
      HQ02 : Struct   // Filtereinheit
         Niv_Leckage : Bool;   // BL12
         GW_p_FG : Bool;   // BP02
         S_FG_zu : Bool;   // BG09
         S_Dkl_FG_li : Bool;   // BG10
         S_Dkl_FG_re : Bool;   // BG1
         Quitt_FW : Bool;
         Quitt_FW_erlaubt : Bool;
         WarnGr_FW : Real;
         Wechsel_FW : Real;
      END_STRUCT;
      GP01 : Struct   // HF-Versorgung
         Versorgung : Bool;
         Entsorgung : Bool;
         Niv_leer : Bool;   // BL17
         Niv_max : Bool;   // BL20
         IBC_vorhanden : Bool;   // BG21
         Tür_zu_vorn : Bool;   // BG44
         Tür_zu_seitlich : Bool;   // BG43
         LS_PuSu : Bool;   // BL18
         LS_Pumpe : Bool;   // BL15
         LS_Doppelrohr_BL19 : Bool;   // BL19
         LS_PFA_Übergang : Bool;   // BL16
         LS_Uml_Tunnel : Bool;   // BL34
         Niv_Proz : USInt;
         Status : USInt;
      END_STRUCT;
      GP02 : Struct   // HF-Entsorgung
         Versorgung : Bool;
         Entsorgung : Bool;
         Niv_leer : Bool;   // BL24
         Niv_max : Bool;   // BL23
         IBC_vorhanden : Bool;   // BG22
         Tür_zu_seitlich : Bool;   // BG45
         LS_PuSu : Bool;   // BL18
         LS_Pumpe : Bool;   // BL27
         LS_PFA_Übergang : Bool;   // BL25
         LS_Doppelrohr_BL26 : Bool;   // BL26
         LS_Doppelschlauch_BL32 : Bool;   // BL32
         LS_Doppelschlauch_BL33 : Bool;   // BL33
         Niv_Proz : USInt;
         Status : USInt;
      END_STRUCT;
      Havarie_GP0x : Struct
         Soll_Spuelen_CM0x : Real;   // [l]
         Ist_Spuelen_CM0x : Real;   // [l]
      END_STRUCT;
      CL0x : Struct
         "LS_CL01.BL28" : Bool;   // Leckage OK Übergabestation CL01 CL01.BL28
         "LS_CL02.BL29" : Bool;   // Leckage OK Pumpensumpf Säurebecken CL02 CL02.BL29
         Niv_Proz_CL01 : USInt;
         Niv_Proz_CL02 : USInt;
      END_STRUCT;
      FP_CM01 : Struct   // GP01
         Ein : Bool;
         Auto : Bool;
         Bedienung_Erlaubt : Bool;
         betriebsbereit : Bool;
         Stoerung : Bool;
         Sp_Ventil : Struct
            Sollzeit : Int;   // [s]
            Restzeit : Int;   // [s]
         END_STRUCT;
         Sp_Filter : Struct
            Zeit_leeren_Saure : Int;   // [s]
            Zeit_leeren_CM05 : Int;
            Zeit_Spülen : Int;   // [s]
            Wartezeit : Int;   // [s]
            Zeit_füllen : Int;   // [s]
            Restzeit : Int;   // [s]
         END_STRUCT;
         Drucktest_Pumpe : Struct
            Solldruck : Real;
            Sollzeit : Int;
            Restzeit : Int;
            Schritt : USInt;
         END_STRUCT;
         Drucktest_Filter : Struct
            Solldruck : Real;
            Sollzeit : Int;
            Restzeit : Int;
            Schritt : USInt;
         END_STRUCT;
         BA : USInt;   // 0=normal, 1=Filterwechsel, 2=Spülen
         Status : USInt;
         Status_FW : USInt;
         SW_Hand : Int;   // [%]
         SW_Auto_AZ : Int;   // [%]
         SW_Auto_aAZ : Int;   // [%]
         speed : Int;   // [%]
      END_STRUCT;
      UP_CM01 : Struct   // GP02
         Ein : Bool;
         Auto : Bool;
         Bedienung_Erlaubt : Bool;
         betriebsbereit : Bool;
         Stoerung : Bool;
         Sp_Ventil : Struct
            Sollzeit : Int;   // [s]
            Restzeit : Int;   // [s]
         END_STRUCT;
         Drucktest : Struct
            Solldruck : Real;
            Sollzeit : Int;
            Restzeit : Int;
            Schritt : USInt;
         END_STRUCT;
         BA : USInt;   // 0=normal, 1=Ents GP02, 2= Ents GP01, 3=Ents. CM05, 4=Spülen
         Status : USInt;
         SW_Hand : Int;   // [%]
         SW_Auto_AZ : Int;   // [%]
         SW_Auto_aAZ : Int;   // [%]
         speed : Int;   // [%]
      END_STRUCT;
      UP_CM03 : Struct   // GP03
         Ein : Bool;
         Auto : Bool;
         betriebsbereit : Bool;
         Bedienung_Erlaubt : Bool;
         Stoerung : Bool;
         Sp_Ventil : Struct
            Sollzeit : Int;   // [s]
            Restzeit : Int;   // [s]
         END_STRUCT;
         Drucktest : Struct
            Solldruck : Real;
            Sollzeit : Int;
            Restzeit : Int;
            Schritt : USInt;
         END_STRUCT;
         BA : USInt;   // 0=normal, 1=Ents. CM05, 2=Spülen
         Status : USInt;
         SW_Hand : Int;   // [%]
         SW_Auto_AZ : Int;   // [%]
         SW_Auto_aAZ : Int;   // [%]
         speed : Int;   // [%]
      END_STRUCT;
      FP_CM02 : Struct   // GP04
         Ein : Bool;
         Auto : Bool;
         Bedienung_Erlaubt : Bool;
         betriebsbereit : Bool;
         Stoerung : Bool;
         Sp_Ventil : Struct
            Sollzeit : Int;   // [s]
            Restzeit : Int;   // [s]
         END_STRUCT;
         Sp_Filter : Struct
            Zeit_leeren_Saure : Int;   // [s]
            Zeit_leeren_CM05 : Int;
            Zeit_Spülen : Int;   // [s]
            Wartezeit : Int;   // [s]
            Zeit_füllen : Int;   // [s]
            Restzeit : Int;   // [s]
         END_STRUCT;
         Drucktest_Pumpe : Struct
            Solldruck : Real;
            Sollzeit : Int;
            Restzeit : Int;
            Schritt : USInt;
         END_STRUCT;
         Drucktest_Filter : Struct
            Solldruck : Real;
            Sollzeit : Int;
            Restzeit : Int;
            Schritt : USInt;
         END_STRUCT;
         BA : USInt;   // 0=normal, 1=Filterwechse, 2=Spülen
         Status : USInt;
         Status_FW : USInt;
         SW_Hand : Int;   // [%]
         SW_Auto_AZ : Int;   // [%]
         SW_Auto_aAZ : Int;   // [%]
         speed : Int;   // [%]
      END_STRUCT;
      UP_CM02 : Struct   // GP05
         Ein : Bool;
         Auto : Bool;
         Bedienung_Erlaubt : Bool;
         betriebsbereit : Bool;
         Stoerung : Bool;
         Sp_Ventil : Struct
            Sollzeit : Int;   // [s]
            Restzeit : Int;   // [s]
         END_STRUCT;
         Drucktest : Struct
            Solldruck : Real;
            Sollzeit : Int;
            Restzeit : Int;
            Schritt : USInt;
         END_STRUCT;
         BA : USInt;   // 0=normal, 1=Ents GP02, 2= Ents GP01, 3=Ents. CM05, 4=Spülen
         Status : USInt;
         SW_Hand : Int;   // [%]
         SW_Auto_AZ : Int;   // [%]
         SW_Auto_aAZ : Int;   // [%]
         speed : Int;   // [%]
      END_STRUCT;
      UP_CM04 : Struct   // GP06
         Ein : Bool;
         Auto : Bool;
         betriebsbereit : Bool;
         Bedienung_Erlaubt : Bool;
         Stoerung : Bool;
         Sp_Ventil : Struct
            Sollzeit : Int;   // [s]
            Restzeit : Int;   // [s]
         END_STRUCT;
         Drucktest : Struct
            Solldruck : Real;
            Sollzeit : Int;
            Restzeit : Int;
            Schritt : USInt;
         END_STRUCT;
         BA : USInt;   // 0=normal, 1=Ents. CM05, 2=Spülen
         Status : USInt;
         SW_Hand : Int;   // [%]
         SW_Auto_AZ : Int;   // [%]
         SW_Auto_aAZ : Int;   // [%]
         speed : Int;   // [%]
      END_STRUCT;
      Pu_CM05 : Struct   // GP11
         Ein : Bool;
         Auto : Bool;
         Bedienung_Erlaubt : Bool;
         Sp_Ventil : Struct
            Sollzeit : Int;   // [s]
            Restzeit : Int;   // [s]
         END_STRUCT;
         Drucktest : Struct
            Solldruck : Real;
            Sollzeit : Int;
            Restzeit : Int;
            Schritt : USInt;
         END_STRUCT;
         BA : USInt;   // 0=Entl., 1=Kreislauf, 2=Spülen
         Status : USInt;
      END_STRUCT;
      Pu_CL01 : Struct   // GP08
         Ein : Bool;
         Auto : Bool;
         Bedienung_Erlaubt : Bool;
         Sp_Ventil : Struct
            Sollzeit : Int;   // [s]
            Restzeit : Int;   // [s]
         END_STRUCT;
         BA : USInt;   // 0=Ents. CM05, 1=Spülen
         Status : USInt;
      END_STRUCT;
      Pu_CL02 : Struct   // GP09
         Ein : Bool;
         Auto : Bool;
         Bedienung_Erlaubt : Bool;
         Sp_Ventil : Struct
            Sollzeit : Int;   // [s]
            Restzeit : Int;   // [s]
         END_STRUCT;
         BA : USInt;   // 0=Ents. CM05, 1=Spülen
         Status : USInt;
      END_STRUCT;
      Pu_Entl_GP01 : Struct   // GP12
         Ein : Bool;
         Auto : Bool;
         Bedienung_Erlaubt : Bool;
         Sp_Ventil : Struct
            Sollzeit : Int;   // [s]
            Restzeit : Int;   // [s]
         END_STRUCT;
         BA : USInt;   // 0=Ents. CM05, 1=Spülen
         Status : USInt;
      END_STRUCT;
      Pu_Vers_GP01 : Struct   // GP13
         Ein : Bool;
         Auto : Bool;
         Bedienung_Erlaubt : Bool;
         Sp_Ventil : Struct
            Sollzeit : Int;   // [s]
            Restzeit : Int;   // [s]
         END_STRUCT;
         BA : USInt;   // 0=Vers UVGP01, 1=Ents CM05, 2=Spülen
         Status : USInt;
      END_STRUCT;
      Pu_Entl_GP02 : Struct   // GP07
         Ein : Bool;
         Auto : Bool;
         Bedienung_Erlaubt : Bool;
         Sp_Ventil : Struct
            Sollzeit : Int;   // [s]
            Restzeit : Int;   // [s]
         END_STRUCT;
         BA : USInt;   // 0=Ents. CM05, 1=Spülen
         Status : USInt;
      END_STRUCT;
      Pu_Vers_GP02 : Struct   // GP10
         Ein : Bool;
         Auto : Bool;
         Bedienung_Erlaubt : Bool;
         Sp_Ventil : Struct
            Sollzeit : Int;   // [s]
            Restzeit : Int;   // [s]
         END_STRUCT;
         BA : USInt;   // 0=Vers UVGP01, 1=Ents CM05,2= Spülen
         Status : USInt;
      END_STRUCT;
      Pu_Entleeren : Struct   // GP14
         Ein : Bool;
         Status : USInt;
      END_STRUCT;
      Ventil : Struct   // 0 = Aus, 1= aktiv, 2=Störung
         "CM01.QM18" : USInt;   // Eingang Saugleitung Filterpumpe GP01 Säure 01 CM01.QM18
         "CM01.QM19" : USInt;   // Eingang Spülleitung Filterpumpe GP01 Säure 01 CM01.QM19
         "CM01.QM20" : USInt;   // Eingang Spülleitung Umwälzpumpe GP02 Säure 01 CM01.QM20
         "HQ01.QM21" : USInt;   // EingangSäureleitung Filtereinheit HQ02 Säure 01 CM01.QM21
         "HQ01.LV01" : USInt;   // Entlüftungs-/ Überdruckventil Beutelfilter Säure 01 HQ01.LV01
         "HQ01.QM22" : USInt;   // Eingang Spülleitung Filtereinheit HQ01 Säure 01 HQ01.QM22
         "HQ01.QM23" : USInt;   // Ausgang Säureleitung Filtereinheit HQ01 Säure 01 HQ01.QM23
         "HQ01.QM24" : USInt;   // Ausgang Spülleitung Filtereinheit HQ01 Säure 01 zu Sammeltank HQ01.QM24
         "CM01.QM25" : USInt;   // Eingang Saugleitung Umwälzpumpe GP02 Säure 01 CM01.QM25
         "CM01.QM26" : USInt;   // Ausgang Druckleitung Umwälzpumpe GP02 Säure 01 CM01.QM26
         "CM01.QM27" : USInt;   // Ausgang Spülleitung Umwälzpumpe GP02 Säure 01 zu Sammeltank CM01.QM27
         "CM03.QM33" : USInt;   // Eingang Saugleitung Umwälzpumpe GP03 Spülbecken 1 CM03.QM33
         "CM03.QM34" : USInt;   // Ausgang Druckleitung Umwälzpumpe GP03 Spülbecken 1 CM03.QM34
         "CM03.QM36" : USInt;   // Eingang Spülleitung Umwälzpumpe GP03 Spülbecken 1 CM03.QM36
         "CM03.QM37" : USInt;   // Ausgang Spülleitung Umwälzpumpe GP03 Spülbecken 1 CM03.QM37
         "CM02.QM55" : USInt;   // Eingang Saugleitung Filterpumpe GP04 Säure 02 CM02.QM55
         "CM02.QM56" : USInt;   // Eingang Spülleitung Filterpumpe GP04 Säure 02 CM02.QM56
         "CM02.QM57" : USInt;   // Eingang Spülleitung Umwälzpumpe GP05 Säure 02 CM02.QM57
         "HQ02.QM58" : USInt;   // Eingang Spülleitung Filtereinheit HQ02 Säure 02 CM02.QM58
         "HQ02.LV02" : USInt;   // Entlüftungs-/ Überdruckventil Beutelfilter Säure 02 HQ02.LV02
         "HQ02.QM59" : USInt;   // Eingang Säureleitung Filtereinheit HQ02 Säure 02 HQ02.QM59
         "HQ02.QM60" : USInt;   // Ausgang Säureleitung Filtereinheit HQ02 Säure 02 HQ02.QM60
         "HQ02.QM61" : USInt;   // Ausgang Spülleitung Filtereinheit HQ02 Säure 02 zu Sammeltank HQ02.QM61
         "CM02.QM62" : USInt;   // Eingang Saugleitung Umwälzpumpe GP05 Säure 02 CM02.QM62
         "CM02.QM63" : USInt;   // Ausgang Druckleitung Umwälzpumpe GP05 Säure 02 CM02.QM63
         "CM02.QM64" : USInt;   // Ausgang Spülleitung Umwälzpumpe GP05 Säure 02 zu Sammeltank CM02.QM64
         "CM04.QM72" : USInt;   // Eingang Saugleitung Umwälzpumpe GP06 Spülbecken 2 CM04.QM72
         "CM04.QM73" : USInt;   // Ausgang Druckleitung Umwälzpumpe GP06 Spülbecken 2 CM04.QM73
         "CM04.QM75" : USInt;   // Eingang Spülleitung Umwälzpumpe GP06 Spülbecken 2 CM04.QM75
         "CM04.QM76" : USInt;   // Ausgang Spülleitung Umwälzpumpe GP06 Spülbecken 2 CM04.QM76
         "CM04.QM77" : USInt;   // Frischwasserzufuhr Nachdosierung Spülbecken 2 CM04.QM77
         "CL01.QM51" : USInt;   // Zuleitung VE-Wasser-Spülung Pumpe GP08 CL01.QM51
         "CL02.QM52" : USInt;   // Zuleitung VE-Wasser-Spülung Pumpe GP09 CL02.QM52
         "CM05.QM61" : USInt;   // Saugseite Förderpumpe Entleerung GP11 Sammeltank CM05 CM05.QM61
         "CM05.QM62" : USInt;   // Eingang Spülleitung Förderpumpe GP11 Sammeltank CM05 CM05.QM62
         "CM05.QM63" : USInt;   // Ausgang Spülleitung Förderpumpe GP11 Sammeltank CM05 CM05.QM63
         "CM05.QM64" : USInt;   // Druckseite Förderpumpe Entleerung GP11 Sammeltank CM05 CM05.QM64
         "CM03.QM35" : USInt;   // VE-Wasserleitung Spritzregister Spülbecken 1 CM03.QM35
         "CM04.QM74" : USInt;   // VE-Wasserleitung Spritzregister Spülbecken 2 CM04.QM74
         "GP01.QM14" : USInt;   // PFA Schlauchleitung Anbindung IBC Quick Connect Entsorgung GP01.QM14
         "GP01.QM15" : USInt;   // Eingang Saugleitung Membranpumpe GP13 Versorgung Frischsäure GP01.QM15
         "GP01.QM16" : USInt;   // Eingang Spülleitung Membranpumpe GP13 Versorgung Frischsäure GP01.QM16
         "GP01.QM17" : USInt;   // Ausgang Spülleitung Membranpumpe GP13 Versorgung zu Sammeltank GP01.QM17
         "GP01.QM18" : USInt;   // Ausgang Druckleitung Membranpumpe GP13 Versorgung zu UV-GP01 GP01.QM18
         "GP01.QM19" : USInt;   // Verriegelung UV-GP01 Versorgungsleitung zu Säure CM2 GP01.QM19
         "GP01.QM20" : USInt;   // Verriegelung UV-GP01 Versorgungsleitung zu Säure CM1 GP01.QM20
         "GP01.QM21" : USInt;   // Verriegelung UV-GP01 Versorgungsleitung zur Entsorgung GP02 GP01.QM21
         "GP01.QM22" : USInt;   // Verriegelung UV-GP01 Versorgungsleitung zur Versorgung GP01 GP01.QM22
         "GP01.QM23" : USInt;   // VE-Wasser-Spülung GP12 zu Auffangwanne GP01.QM23
         "GP02.QM37" : USInt;   // VE-Wasser-Ventil Leckagesumpf Entsorgung Altsäure GP02.QM37
         "GP02.QM38" : USInt;   // Eingang Saugleitung Membranpumpe GP10 Versorgung aus GP02 GP02.QM38
         "GP02.QM39" : USInt;   // Eingang Spülleitung Membranpumpe GP10 Versorgung aus GP02 GP02.QM39
         "GP02.QM40" : USInt;   // Ausgang Druckleitung Membranpumpe GP10 zu Sammeltank CM05 GP02.QM40
         "GP02.QM41" : USInt;   // Verriegelung UV-GP02 Versorgungsleitung zu UV-GP01 GP02.QM41
         "GP02.QM42" : USInt;   // Ausgang Spülleitung Membranpumpe GP10 zu Sammeltank CM05 GP02.QM42
         "GP02.QM43" : USInt;   // Verriegelung UV-GP02 Entsorgungsleitung zu Entsorgung GP02 GP02.QM43
         "GP02.QM44" : USInt;   // Verriegelung UV-GP02 Entsorgungsleitung zu Versorgung GP01 GP02.QM44
         "GP02.QM45" : USInt;   // Verriegelung UV-GP02 Entsorgungsleitung von Säurebecken CM01 GP02.QM45
         "GP02.QM46" : USInt;   // Verriegelung UV-GP02 Entsorgungsleitung von Säurebecken CM02 GP02.QM46
      END_STRUCT;
      Betriebsart : Struct
         Tipp : Bool;
         Hand : Bool;
         Automatik : Bool;
         Anzeige : USInt;
      END_STRUCT;
      QF : Struct
         WR02 : Struct
            Auto : Bool;
            Hand : Bool;
            Tipp : Bool;
            T_einfahren : Bool;
            T_ausfahren : Bool;
            S_Pos_Ue : Bool;
            S_Pos_BE : Bool;
            S_BK_vl : Bool;
            S_BK_vr : Bool;
            S_BK_hl : Bool;
            S_BK_hr : Bool;
            A_einfahren : Bool;
            A_ausfahren : Bool;
         END_STRUCT;
         WR03 : Struct
            Auto : Bool;
            Hand : Bool;
            Tipp : Bool;
            T_einfahren : Bool;
            T_ausfahren : Bool;
            S_Pos_Ue : Bool;
            S_Pos_BE : Bool;
            S_BK_vl : Bool;
            S_BK_vr : Bool;
            S_BK_hl : Bool;
            S_BK_hr : Bool;
            A_einfahren : Bool;
            A_ausfahren : Bool;
         END_STRUCT;
         P25_kurz_fertig : Bool;
         P25_lang_fertig : Bool;
         P26_fertig : Bool;
         P27_fertig : Bool;
         P28_fertig : Bool;
         P29_kurz_fertig : Bool;
         P29_lang_fertig : Bool;
         P30_fertig : Bool;
      END_STRUCT;
      TW : Struct
         Knauf_Auto : Bool;
         T_Halt : Bool;
         T_vor : Bool;
         T_rueck : Bool;
         T_heben : Bool;
         T_senken : Bool;
         T_heben_li : Bool;
         T_senken_li : Bool;
         T_heben_re : Bool;
         T_senken_re : Bool;
      END_STRUCT;
      Aufgabe : Struct
         Anf_GO : Bool;   // Beide QF nach aussen
         Freigabe : Bool;   // Datenübernahme
         KS_vl_erlaubt : Bool;   // B/E 1
         KS_vr_erlaubt : Bool;   // B/E 2
         GO_li_erlaubt : Bool;   // B/E 3
         GO_re_erlaubt : Bool;   // B/E 4
         KS_hl_erlaubt : Bool;   // B/E 5
         KS_hr_erlaubt : Bool;   // B/E 6
         LS_v_erlaubt : Bool;   // B/E 1
         LS_h_erlaubt : Bool;   // B/E 5
      END_STRUCT;
      Betriebsmodus : Struct
         Normal : Bool;
         Kombi : Bool;
         Wechsel_erlaubt : Bool;
         Korb_151 : Bool;
         Korb_161 : Bool;
         Anzeige : USInt;
      END_STRUCT;
   END_VAR
BEGIN
END_DATA_BLOCK

DATA_BLOCK "DB_Fahr-Hubzeit"   // DB5
{ S7_Optimized_Access := 'FALSE' }
// stored: AutoNumber false
   VAR RETAIN
      FZ_Typ_Pos : Real := 1.0;   // Fahrzeit typisch Position zu Position
      FZ_Typ_Halt : Real := 5.0;   // Fahrzeit typisch für Positionierung
      UZ_typ : Real := 40.0;   // typische Umsetzzeit (für Zwischenschieben)
      HZ_Gestell_langsam : Real := 20.0;   // Hubzeit typisch für Gestelle bei langsamen Hub
      HZ_Gestell_schnell : Real := 15.0;   // Hubzeit typisch für Gestelle bei schnellen Hub
      HZ_Trommel_langsam : Real := 20.0;   // Hubzeit typisch für Trommeln bei langsamen Hub
      HZ_Trommel_schnell : Real := 15.0;   // Hubzeit typisch für Trommeln bei schnellen Hub
      SZ_Gestell_langsam : Real := 20.0;   // Senkzeit typisch für Gestelle bei langsamen Hub
      SZ_Gestell_schnell : Real := 15.0;   // Senkzeit typisch für Gestelle bei schnellen Hub
      SZ_Trommel_langsam : Real := 20.0;   // Senkzeit typisch für Trommeln bei langsamen Hub
      SZ_Trommel_schnell : Real := 15.0;   // Senkzeit typisch für Trommeln bei schnellen Hub
      TS_Zeit : Real := 0.0;   // Schwenkzeit Tropfwanne typisch
   END_VAR
BEGIN
END_DATA_BLOCK

DATA_BLOCK "DB_GroupConfig"   // DB42
{ S7_Optimized_Access := 'FALSE' }
// stored: AutoNumber false
   VAR RETAIN
      AnzGroup : Int := 0;   // + Anzahl der Definierten Gruppen (wird mit FW-Editor eingetragen)
      OffsetAdr : Int := 10;   // * Adresse der ersten Gruppendefinition
      resW : Int := 0;
      resD1 : DInt := 0;
      Gruppe : Array[0..9] of Struct   // * Feldlänge anpassen (Inhalte werden mit FW-Editor erzeugt)
         Start : Int;   // + Startadresse in Byte der Gruppe in diesem DB sieh Def
         QT_Nr : Int;   // + zu benutzender Quertransport, wenn reihenübergreifende Gruppe
         Skip_enable : Bool;   // + Überspringen möglich
         OptiGroup : Bool;   // + Optimierungsberechnung berücksichtigen
         Vorzugsreihe : Bool;   // + Vorzugsweise innerhalb der gleichen Reihe umsetzen
         res3 : Bool;
         res4 : Bool;
         res5 : Bool;
         res6 : Bool;
         res7 : Bool;
         res8 : Bool;
         res9 : Bool;
         res10 : Bool;
         res11 : Bool;
         res12 : Bool;
         res13 : Bool;
         res14 : Bool;
         res15 : Bool;
      END_STRUCT;
      Def : Array[1..10] of Byte;   // * Definition der Gruppen-Positionen
   END_VAR
BEGIN
   Gruppe[0..9].Start := 0;
   Gruppe[0..9].QT_Nr := 0;
   Gruppe[0..9].Skip_enable := FALSE;
   Gruppe[0..9].OptiGroup := FALSE;
   Gruppe[0..9].Vorzugsreihe := FALSE;
   Gruppe[0..9].res3 := FALSE;
   Gruppe[0..9].res4 := FALSE;
   Gruppe[0..9].res5 := FALSE;
   Gruppe[0..9].res6 := FALSE;
   Gruppe[0..9].res7 := FALSE;
   Gruppe[0..9].res8 := FALSE;
   Gruppe[0..9].res9 := FALSE;
   Gruppe[0..9].res10 := FALSE;
   Gruppe[0..9].res11 := FALSE;
   Gruppe[0..9].res12 := FALSE;
   Gruppe[0..9].res13 := FALSE;
   Gruppe[0..9].res14 := FALSE;
   Gruppe[0..9].res15 := FALSE;
   Def[1..10] := 16#00;
END_DATA_BLOCK

DATA_BLOCK "DB_HW"   // DB53
{ S7_Optimized_Access := 'FALSE' }
// stored: AutoNumber false
   VAR RETAIN
      Anzahl : Int := 0;   // * Anzahl der Höhenwechsel
      Offset : Int := 10;   // * Startadresse Einträge
      lengHW : Int := 6;   // * Länge eines Eintrages in Byte
      resW : Int := 0;
      resW1 : Int := 0;
      HW : Array[1..8] of Struct
         Pos : DInt;
         Ebene_rck : Byte;
         Ebene_vor : Byte;
      END_STRUCT;
   END_VAR
BEGIN
   HW[1..8].Pos := 0;
   HW[1..8].Ebene_rck := 16#00;
   HW[1..8].Ebene_vor := 16#00;
END_DATA_BLOCK

DATA_BLOCK "DB_Korbumlaeufe"   // DB330
{ S7_Optimized_Access := 'TRUE' }
// stored: AutoNumber false, MemoryReserve 100
   VAR RETAIN
      Korb : Array[1..28] of Struct
         Durchlaeufe : Int;
         max_Durchlaeufe : Int;
         Warnung : Bool;
         max_erreicht : Bool;
      END_STRUCT;
   END_VAR
BEGIN
   Korb[1..13].max_Durchlaeufe := 15;
END_DATA_BLOCK

DATA_BLOCK "DB_KorrPos"   // DB54
{ S7_Optimized_Access := 'FALSE' }
// stored: AutoNumber false
   VAR RETAIN
      Offset : Int := 10;   // Beginn erste Struktur
      Leng : Int := 200;   // Länge einer Struktur
      resI : Int := 0;
      Berechnung_ein : Bool := FALSE;   // * Berechnung durchführen
      res : Bool := FALSE;
      res1 : Bool := FALSE;
      res2 : Bool := FALSE;
      res3 : Bool := FALSE;
      res4 : Bool := FALSE;
      res5 : Bool := FALSE;
      res6 : Bool := FALSE;
      resB : Byte := 16#00;
      resI1 : Int := 0;
      TW : Array[1..10] of Struct
         Pos : Array[1..100] of Int;
      END_STRUCT;
   END_VAR
BEGIN
   TW[1].Pos[1..100] := 0;
   TW[2].Pos[1..100] := 0;
   TW[3].Pos[1..100] := 0;
   TW[4].Pos[1..100] := 0;
   TW[5].Pos[1..100] := 0;
   TW[6].Pos[1..100] := 0;
   TW[7].Pos[1..100] := 0;
   TW[8].Pos[1..100] := 0;
   TW[9].Pos[1..100] := 0;
   TW[10].Pos[1..100] := 0;
END_DATA_BLOCK

DATA_BLOCK "DB_Optimierung_HCA"   // DB170
{ S7_Optimized_Access := 'TRUE' }
// stored: AutoNumber false, MemoryReserve 100
   VAR
      Restzeit_Kurz_Links { ExternalWritable := 'False'} : DInt;
      Restzeit_Kurz_Rechts { ExternalWritable := 'False'} : DInt;
      Restzeit_Lang { ExternalWritable := 'False'} : DInt;
      Restzeit_Gross_Links { ExternalWritable := 'False'} : DInt;
      Restzeit_Gross_Rechts { ExternalWritable := 'False'} : DInt;
      Restzeit { ExternalAccessible := 'False'; ExternalVisible := 'False'; ExternalWritable := 'False'} : Array[1..18] of DInt;
   END_VAR
BEGIN
END_DATA_BLOCK

DATA_BLOCK "DB_PAR_ID"   // DB55
{ S7_Optimized_Access := 'FALSE' }
AUTHOR : MS
// stored: AutoNumber false
   VAR RETAIN
      Anz : Int := 0;
      Offset : Int := 50;   // * Beginn Daten
      Leng : Int := 10;   // * Länge Daten
      resd : DWord := 16#0000_0000;
      resd1 : DWord := 16#0000_0000;
      resd2 : DWord := 16#0000_0000;
      resd3 : DWord := 16#0000_0000;
      resd4 : DWord := 16#0000_0000;
      resd5 : DWord := 16#0000_0000;
      resd6 : DWord := 16#0000_0000;
      resd7 : DWord := 16#0000_0000;
      resd8 : DWord := 16#0000_0000;
      resd9 : DWord := 16#0000_0000;
      resd10 : DWord := 16#0000_0000;
      Par_Config : Array[1..30] of Struct   // * Feldlänge anpassen Anzahl Positionen
         PAR1 : Byte;   // Beginn
         PAR2 : Byte;
         PAR3 : Byte;
         PAR4 : Byte;
         PAR5 : Byte;
         PAR6 : Byte;
         PAR7 : Byte;
         PAR8 : Byte;
         PAR9 : Byte;
         PAR10 : Byte;
      END_STRUCT;
   END_VAR
BEGIN
   Par_Config[1..24].PAR1 := 16#01;
   Par_Config[25..30].PAR1 := 16#00;
   Par_Config[1..30].PAR2 := 16#00;
   Par_Config[1..30].PAR3 := 16#00;
   Par_Config[1..30].PAR4 := 16#00;
   Par_Config[1..30].PAR5 := 16#00;
   Par_Config[1..30].PAR6 := 16#00;
   Par_Config[1..30].PAR7 := 16#00;
   Par_Config[1..30].PAR8 := 16#00;
   Par_Config[1..30].PAR9 := 16#00;
   Par_Config[1..30].PAR10 := 16#00;
END_DATA_BLOCK

DATA_BLOCK "DB_POS"   // DB51
{ S7_Optimized_Access := 'FALSE' }
AUTHOR : MS
// stored: AutoNumber false
   VAR RETAIN
      ANZAHL : Int := 58;   // Anzahl der Positionen
      Offset : Int := 50;   // * Beginn der Datenstruktur
      LENG : Int := 100;   // * Länge einer Position in Byte
      akt_POS : Int := 13;   // Position in Bearbeitung
      resW : Int := 0;
      resDW1 : DWord := 16#0000_0000;
      RESDW2 : DWord := 16#0000_0000;
      RESDW3 : DWord := 16#0000_0000;
      RESDW4 : DWord := 16#0000_0000;
      RESDW5 : DWord := 16#0000_0000;
      RESDW6 : DWord := 16#0000_0000;
      RESDW7 : DWord := 16#0000_0000;
      RESDW8 : DWord := 16#0000_0000;
      RESDW9 : DWord := 16#0000_0000;
      RESDW10 : DWord := 16#0000_0000;
      POS : Array[0..30] of Struct   // * Feldlänge anpassen
         Typ : Byte;   // Badtyp 0=Anlagenpos normal, 1-3=Be-Entladestand, 5=Speicher ,10=QT-Pos, 255 Dum
         SubTyp : Byte;   // Untertyp der Position 5=ExpoVorruf ignorieren bei 2xEinsetzen, 1=Sperre bei Alt
         Prio_Pos : Byte;   // Priorität des Bades (höchste Priorität==0
         SchiebePos : Byte;   // Position auf die FW geschoben wird, wenn er ohne Befehl hier steht
         Reihe : Byte;   // Reihe auf der sich die Position befindet
         FW_Nr : Byte;   // FW_Nr des FW, der über dieser Pos ist
         Optipos : Bool;   // WT wird in die Optimierungsrechnung einbezogen
         berechnet : Bool;   // WT wurde von der Optimierung berechnet
         Quelle : Bool;   // Position ist als Quelle reserviert
         Ziel : Bool;   // Position ist als Ziel reserviert
         FW_kommt : Bool;   // FW will dieses Bad überfahren
         FW_in_POS : Bool;   // Fahrwagen über Bad positioniert
         FW_Hebt : Bool;   // Fahrwagen hebt aus
         FW_Senkt : Bool;   // Fahrwagen setzt ein
         Sperre_in : Bool;   // Bad Einfahrsperre
         Sperre_FW : Bool;   // Bad Überfahrsperre
         Sperre_out : Bool;   // Bad Ausfahrsperre
         IN_OUT_nen : Bool;   // Einsetzen bzw. Ausheben nicht möglich, da Warenbewegung oder Deckel zu usw.
         lngsm_IN : Bool;   // langsames Einsetzen erforderlich-abhängig von immer_schnell
         lngsm_OUT : Bool;   // langsames Ausheben erforderlich-abhängig von immer_schnell
         immer_schnell : Bool;   // trockene Position (keine ATZ, schneller Hub erlaubt)
         QT_reserviert : Bool;   // Position ist durch QT reserviert
         KS_erlaubt : Bool;   // Pos darf mit KS befülltwerden
         LS_erlaubt : Bool;   // Pos darf mit LS befüllt werden
         GO_erlaubt : Bool;   // Pos darf mit GO befüllt werden
         Belegt_KS : Bool;   // Belegt mit KS
         Belegt_LS : Bool;   // Belegt mit LS
         Belegt_GO : Bool;   // Belegtmit GO
         Spr_Off : Bool;   // Oberhalb Z nicht spritzen
         Opt_Abgelehnt : Bool;   // Einfahrt durch Opti abgelehnt
         notFG_out : Bool;   // Position darf nicht geräumt werden (Merkersystem)
         notFG_in : Bool;   // Position darf nicht befüllt werden (Merkersystem)
         Anmeldung : Bool;   // bevorzugte Behandlung anmelden
         fPosfree : Bool;   // Folgeposition muß frei sein
         QT_Sperre : Bool;   // Position ist durch QT gesperrt FW darf Pos nicht bedienen
         Vorsperre : Bool;   // Einfahrsperre anmelden
         QT_FW_Ruf : Bool;   // QT wird auf dieser Position von einem FW benötigt
         QT_ext_Ruf : Bool;   // QT wird auf dieser Position von einem externen Gerät benötigt
         Bef_ende : Bool;   // in diesem Bad muß der Befehlsindex geschaltet werden
         DoppelTauch : Bool;   // Doppeltauchen angefordert
         ignor_Exp : Bool;   // Expozeit ignorieren (Transport)
         ignor_ESp : Bool;   // ignoriere Einfahrsperre (notFG_in)
         ignor_fPosFree : Bool;   // ignoriere fPosFree (z.B. für Freigabe Pos kurz vor Expoende)
         UebergabePos : Bool;   // Übergabe von Wts möglich
         Portable : Bool;   // Im Vorruf und transportierbar
         Checked : Bool;   // Position im ersten Check (FB9) geprüft
         Detailtyp : Byte;   // 0=egal, 11=KS. 12=LS, 20=GO (alleshex)
         BereichsTakte : Byte;   // 0=kein laden, ansonsten auf WTDB.DBB54
         Stand_Nr : Byte;   // Verweis auf Stand Nr
         Absetzhoehe : DInt;   // Absetzhöhe in Inkrementen
         LZ_Nr1 : Byte;   // Verweis auf Ladungszähler Nr1
         LZ_Nr2 : Byte;   // Verweis auf Ladungszähler Nr2
         ZG_1 : Byte;   // Reserve für weitere Verweise
         ZG_2 : Byte;   // Reserve für weitere Verweise
         IncPos : DInt;   // Position des Bades in der Anlage
         IncAbstand_vor : Int;   // min. Abstand zum Bad bei Überfahrsperre
         IncAbstand_rck : Int;   // min. Abstand zum Bad bei Überfahrsperre
         WT_Nr_lang : DInt;   // Warenträger-Nr.
         WT_Stangen_Nr : Byte;   // Stangen-Nr
         WT_DB : Byte;   // DB_Nr Warenstange
         next_WT : Byte;   // WT der sich für diese Pos anmeldet
         Prio : Bool;
         INA : Bool;
         INE : Bool;
         OUTA : Bool;
         OUTE : Bool;
         SpProg : Bool;
         ResAmTW : Bool;
         ResAmQT : Bool;
         Trommel : Bool;   // Kontrolle aktiviert
         Leer_WT : Bool;   // Leerwarenträger HFs aus
         Warnung : Bool;   // in Position wurde eine Warnmeldung ausgelöst
         Alarm : Bool;   // in Position wurde eine Alarmmeldung ausgelöst
         WT_neu : Bool;   // WT wurde vom LZ noch nicht berücksichtigt
         lngsm_Hub : Bool;   // langsam Heben als WT-Parameter
         B_Takte_Null : Bool;   // Bereichstakte sind Null
         enable_reload : Bool;   // laden der Altwerte innerhalb einer Gruppe erlaubt
         WT_Typ : Byte;   // Art des Warenträgers (z.Bsp. bei fester Zuordnung Ware-WT)
         WT_Befx : Int;   // WT Befehlsindex
         Soll_Takte : Int;   // VERWEILTAKTE
         Soll_Expozeit : DInt;   // Sollwert Expositionszeit
         ExpoToleranz : DInt;   // Toleranzwert für Expozeit
         KF_A : Real;   // Korrekturfaktor WT_Auslastung 0..100%-->0..1, Gesamtoberfläche
         KF_Expo : Real;   // Korrekturfaktor Expozeit
         Korr_Restzeit : DInt;   // korregierte Restzeit bis zur Abholung WT
         SonderPos_Offset : DInt;   // Offset für Positionierung außermittig (Höhenwechsel,Blende usw.)
         Restvorsperre : Int;   // Resttakte bis Vorsperre
         Resttakte : Int;   // Taktzähler
         Restzeit : DInt;   // verbleibende Expositionszeit
         Verweilzeit : DInt;   // Verweilzeit
         T_Vorruf : Int;   // Vorrufzeit lößt Vorruf n Sekunden vor Ablauf der Expozeit aus
         T_Pend : Int;   // Auspendelzeit 0..999s
         T_ATZ : Int;   // Abtropfzeit 0..999s
         T_Vorsperre : Int;   // Takte bis Vorsperre zu Sperre wird
         WaitTime : DInt;   // Zeit der Expounterbrechung
         Res_Real : Real;
         belegt : Bool;   // Bad belegt
         Bearbeitung : Bool;   // Badbehandlung läuft
         Vorruf : Bool;   // Bad FW-Vorruf
         fertig : Bool;   // Bad fertig
         AL_Expo : Bool;   // Expotoleranz um 30s überschritten
         Dkl_auf_Pos : Bool;
         Expo_Off : Bool;   // Expozeit unterbrochen (GR-Absenkung)
         yALEX : Bool;   // Alarm Expo auslösen
         US_on_Q : Bool;   // Ultraschall 7s einschalten, wenn Quelle
         AlExp : Bool;   // Alarm Expotoleranz war ein
         MD_Alex : Bool;   // Meldung Expoalarm wurde abgesetzt
         MD_res : Bool;   // Meldung Gleichrichterfehler
         MD_res_1 : Bool;   // Meldung Temperaturreglerfehler
         QT_in_Pos : Bool;   // QT in Position
         res27 : Bool;
         PendHub : Bool;   // Pendelhub aktiv
         Leerzeit : Int;   // Zeit welche Position nicht benutzt
      END_STRUCT;
      RESDW : DWord := 16#0000_0000;
   END_VAR
BEGIN
   POS[0].Typ := 16#00;
   POS[1].Typ := 16#03;
   POS[2..30].Typ := 16#00;
   POS[0..30].SubTyp := 16#00;
   POS[0..30].Prio_Pos := 16#05;
   POS[0..30].SchiebePos := 16#00;
   POS[0..30].Reihe := 16#01;
   POS[0..1].FW_Nr := 16#00;
   POS[2].FW_Nr := 16#01;
   POS[3..10].FW_Nr := 16#00;
   POS[11].FW_Nr := 16#02;
   POS[12..30].FW_Nr := 16#00;
   POS[0..30].Optipos := FALSE;
   POS[0..30].berechnet := FALSE;
   POS[0..30].Quelle := FALSE;
   POS[0..30].Ziel := FALSE;
   POS[0..30].FW_kommt := FALSE;
   POS[0..1].FW_in_POS := FALSE;
   POS[2].FW_in_POS := TRUE;
   POS[3..10].FW_in_POS := FALSE;
   POS[11].FW_in_POS := TRUE;
   POS[12..30].FW_in_POS := FALSE;
   POS[0..30].FW_Hebt := FALSE;
   POS[0..30].FW_Senkt := FALSE;
   POS[0..30].Sperre_in := FALSE;
   POS[0..30].Sperre_FW := FALSE;
   POS[0..30].Sperre_out := FALSE;
   POS[0..30].IN_OUT_nen := FALSE;
   POS[0..30].lngsm_IN := FALSE;
   POS[0..30].lngsm_OUT := FALSE;
   POS[0].immer_schnell := FALSE;
   POS[1..2].immer_schnell := TRUE;
   POS[3..27].immer_schnell := FALSE;
   POS[28].immer_schnell := TRUE;
   POS[29..30].immer_schnell := FALSE;
   POS[0..30].QT_reserviert := FALSE;
   POS[0..30].KS_erlaubt := FALSE;
   POS[0..30].LS_erlaubt := FALSE;
   POS[0..30].GO_erlaubt := FALSE;
   POS[0..30].Belegt_KS := FALSE;
   POS[0..30].Belegt_LS := FALSE;
   POS[0..30].Belegt_GO := FALSE;
   POS[0..30].Spr_Off := FALSE;
   POS[0..30].Opt_Abgelehnt := FALSE;
   POS[0].notFG_out := FALSE;
   POS[1].notFG_out := TRUE;
   POS[2..30].notFG_out := FALSE;
   POS[0].notFG_in := FALSE;
   POS[1].notFG_in := TRUE;
   POS[2..30].notFG_in := FALSE;
   POS[0..30].Anmeldung := FALSE;
   POS[0..30].fPosfree := FALSE;
   POS[0..30].QT_Sperre := FALSE;
   POS[0..30].Vorsperre := FALSE;
   POS[0..30].QT_FW_Ruf := FALSE;
   POS[0..30].QT_ext_Ruf := FALSE;
   POS[0..30].Bef_ende := TRUE;
   POS[0..30].DoppelTauch := FALSE;
   POS[0..30].ignor_Exp := FALSE;
   POS[0..30].ignor_ESp := FALSE;
   POS[0..30].ignor_fPosFree := FALSE;
   POS[0..30].UebergabePos := FALSE;
   POS[0..30].Portable := FALSE;
   POS[0..30].Checked := FALSE;
   POS[0..9].Detailtyp := 16#00;
   POS[10].Detailtyp := 16#16;
   POS[11..12].Detailtyp := 16#00;
   POS[13].Detailtyp := 16#15;
   POS[14].Detailtyp := 16#14;
   POS[15..16].Detailtyp := 16#00;
   POS[17].Detailtyp := 16#13;
   POS[18].Detailtyp := 16#00;
   POS[19].Detailtyp := 16#12;
   POS[20..21].Detailtyp := 16#00;
   POS[22].Detailtyp := 16#11;
   POS[23..30].Detailtyp := 16#00;
   POS[0..30].BereichsTakte := 16#00;
   POS[0].Stand_Nr := 16#00;
   POS[1].Stand_Nr := 16#01;
   POS[2..30].Stand_Nr := 16#00;
   POS[0..30].LZ_Nr1 := 16#00;
   POS[0..30].LZ_Nr2 := 16#00;
   POS[0..30].ZG_1 := 16#00;
   POS[0..30].ZG_2 := 16#00;
   POS[0].IncPos := 12000;
   POS[1].IncPos := 1000;
   POS[2].IncPos := 2000;
   POS[3].IncPos := 3000;
   POS[4].IncPos := 4000;
   POS[5].IncPos := 5000;
   POS[6].IncPos := 6000;
   POS[7].IncPos := 7000;
   POS[8].IncPos := 8000;
   POS[9].IncPos := 9000;
   POS[10].IncPos := 10000;
   POS[11].IncPos := 11000;
   POS[12].IncPos := 12000;
   POS[13].IncPos := 13000;
   POS[14].IncPos := 14000;
   POS[15].IncPos := 15000;
   POS[16].IncPos := 16000;
   POS[17].IncPos := 17000;
   POS[18].IncPos := 18000;
   POS[19].IncPos := 19000;
   POS[20].IncPos := 20000;
   POS[21].IncPos := 21000;
   POS[22].IncPos := 22000;
   POS[23].IncPos := 23000;
   POS[24].IncPos := 24000;
   POS[25].IncPos := 25000;
   POS[26].IncPos := 26000;
   POS[27].IncPos := 27000;
   POS[28].IncPos := 28000;
   POS[29].IncPos := 29000;
   POS[30].IncPos := 30000;
   POS[0].IncAbstand_vor := 0;
   POS[1].IncAbstand_vor := 600;
   POS[2..30].IncAbstand_vor := 0;
   POS[0].IncAbstand_rck := 0;
   POS[1].IncAbstand_rck := 300;
   POS[2..30].IncAbstand_rck := 0;
   POS[0..30].WT_Nr_lang := 0;
   POS[0..30].WT_Stangen_Nr := 16#00;
   POS[0..30].WT_DB := 16#00;
   POS[0..30].next_WT := 16#00;
   POS[0..30].Prio := FALSE;
   POS[0..30].INA := FALSE;
   POS[0..30].INE := FALSE;
   POS[0..30].OUTA := FALSE;
   POS[0..30].OUTE := FALSE;
   POS[0..30].SpProg := FALSE;
   POS[0..30].ResAmTW := FALSE;
   POS[0..30].ResAmQT := FALSE;
   POS[0..30].Trommel := FALSE;
   POS[0..30].Leer_WT := FALSE;
   POS[0..30].Warnung := FALSE;
   POS[0..30].Alarm := FALSE;
   POS[0..30].WT_neu := FALSE;
   POS[0..30].lngsm_Hub := FALSE;
   POS[0..30].B_Takte_Null := FALSE;
   POS[0..3].enable_reload := FALSE;
   POS[4..7].enable_reload := TRUE;
   POS[8..30].enable_reload := FALSE;
   POS[0..30].WT_Typ := 16#00;
   POS[0..30].WT_Befx := 0;
   POS[0..30].Soll_Takte := 0;
   POS[0].Soll_Expozeit := 5;
   POS[1].Soll_Expozeit := 0;
   POS[2].Soll_Expozeit := 360;
   POS[3].Soll_Expozeit := 60;
   POS[4..7].Soll_Expozeit := 1260;
   POS[8..9].Soll_Expozeit := 90;
   POS[10].Soll_Expozeit := 75;
   POS[11..12].Soll_Expozeit := 5;
   POS[13..14].Soll_Expozeit := 75;
   POS[15..16].Soll_Expozeit := 5;
   POS[17].Soll_Expozeit := 75;
   POS[18].Soll_Expozeit := 5;
   POS[19].Soll_Expozeit := 75;
   POS[20].Soll_Expozeit := 5;
   POS[21].Soll_Expozeit := 10;
   POS[22].Soll_Expozeit := 360;
   POS[23..27].Soll_Expozeit := 5;
   POS[28].Soll_Expozeit := 0;
   POS[29..30].Soll_Expozeit := 5;
   POS[0..30].ExpoToleranz := 600;
   POS[0..30].KF_A := 0.0;
   POS[0..30].KF_Expo := 0.0;
   POS[0..30].Korr_Restzeit := 0;
   POS[0..30].SonderPos_Offset := 0;
   POS[0..30].Restvorsperre := 0;
   POS[0..30].Resttakte := 0;
   POS[0..30].Restzeit := 0;
   POS[0..30].Verweilzeit := 0;
   POS[0..30].T_Vorruf := 30;
   POS[0..30].T_Pend := 1;
   POS[0].T_ATZ := 5;
   POS[1..2].T_ATZ := 0;
   POS[3..7].T_ATZ := 10;
   POS[8..9].T_ATZ := 5;
   POS[10].T_ATZ := 10;
   POS[11..12].T_ATZ := 5;
   POS[13..14].T_ATZ := 10;
   POS[15..16].T_ATZ := 5;
   POS[17].T_ATZ := 10;
   POS[18].T_ATZ := 5;
   POS[19].T_ATZ := 10;
   POS[20..21].T_ATZ := 5;
   POS[22].T_ATZ := 10;
   POS[23].T_ATZ := 5;
   POS[24..27].T_ATZ := 2;
   POS[28].T_ATZ := 0;
   POS[29].T_ATZ := 5;
   POS[30].T_ATZ := 2;
   POS[0..30].T_Vorsperre := 0;
   POS[0..30].WaitTime := 0;
   POS[0..30].Res_Real := 0.0;
   POS[0..30].belegt := FALSE;
   POS[0..30].Bearbeitung := FALSE;
   POS[0..30].Vorruf := FALSE;
   POS[0..30].fertig := FALSE;
   POS[0..30].AL_Expo := FALSE;
   POS[0..30].Dkl_auf_Pos := FALSE;
   POS[0..30].Expo_Off := FALSE;
   POS[0..30].yALEX := FALSE;
   POS[0..30].US_on_Q := FALSE;
   POS[0..30].AlExp := FALSE;
   POS[0..30].MD_Alex := FALSE;
   POS[0..30].MD_res := FALSE;
   POS[0..30].MD_res_1 := FALSE;
   POS[0..30].QT_in_Pos := FALSE;
   POS[0..30].res27 := FALSE;
   POS[0].PendHub := TRUE;
   POS[1..2].PendHub := FALSE;
   POS[3].PendHub := TRUE;
   POS[4..10].PendHub := FALSE;
   POS[11..12].PendHub := TRUE;
   POS[13..14].PendHub := FALSE;
   POS[15..16].PendHub := TRUE;
   POS[17].PendHub := FALSE;
   POS[18].PendHub := TRUE;
   POS[19].PendHub := FALSE;
   POS[20..21].PendHub := TRUE;
   POS[22].PendHub := FALSE;
   POS[23].PendHub := TRUE;
   POS[24..30].PendHub := FALSE;
   POS[0..30].Leerzeit := 32767;
END_DATA_BLOCK

DATA_BLOCK "DB_Panel_Posinfo"   // DB52
{ S7_Optimized_Access := 'FALSE' }
// stored: AutoNumber false
   VAR RETAIN
      Offset : Int := 50;   // * Beginn Daten
      Leng : Int := 80;   // * Länge Daten
      resDW1 : DWord := 16#0000_0000;
      resDW2 : DWord := 16#0000_0000;
      resDW3 : DWord := 16#0000_0000;
      resDW4 : DWord := 16#0000_0000;
      last_Takt : DInt := 0;
      Taktzeit : DInt := 0;   // Zeit die der Takt läuft
      Takt_Ware : DInt := 0;   // Zeit seit Ausfahrt letzte Fertigware
      Stop_Anlage : Byte := 16#00;   // ungleich 0-->Kettenbearbeitung anhalten
      Feierabend : Byte := 16#00;   // ungleich 0-->FEIERABENDPROGRAMM
      Sonder_BA : Byte := 16#00;   // ungleich 0-->ELEKTROLYSE, ENTMETALLISIEREN
      IST_Sonder_BA : Byte := 16#00;
      FB_FW_akt : Word := 16#0000;   // an Fernbedienung gewählter FW
      SPS_getaktet : Bool := TRUE;
      resDW10 : DWord := 16#0000_0000;
      resDW11 : DWord := 16#0000_0000;
      resW : Word := 16#0000;
      Pos : Array[1..30] of Struct   // * Feldlänge anpassen
         Prio_Pos : Byte;   // Priorität des Bades (höchste Priorität==0
         lngsm_IN : Bool;   // langsames Einsetzen erforderlich-abhängig von immer_schnell
         lngsm_OUT : Bool;   // langsames Ausheben erforderlich-abhängig von immer_schnell
         res : Bool;
         res1 : Bool;
         res2 : Bool;
         res3 : Bool;
         Luft_Ein : Bool;   // Lufteinblasung ein
         Luft_Auto : Bool;   // Lufteinblasung Automatik
         Verweilzeit : DInt;   // Verweilzeit
         KF_A : Real;   // Korrekturfaktor WT_Auslastung 0..100%-->0..1, Gesamtoberfläche
         KF_Expo : Real;   // Korrekturfaktor Expozeit in %
         T_Vorruf : Int;   // Vorrufzeit lößt Vorruf n Sekunden vor Ablauf der Expozeit aus
         T_Pend : Int;   // Auspendelzeit 0..999s
         T_ATZ : Int;   // Abtropfzeit 0..999s
         NS_Auto : Bool;   // Nachspeisung Automatik
         SR_Auto : Bool;   // Spritzregister Automatik
         res6 : Bool;
         WBE_Ein : Bool;   // Warenbewegung ein
         WBE_Auto : Bool;   // Warenbewegung Automatik
         TS_Pos : Bool;   // Tropfschalenpos.
         res9 : Bool;
         res10 : Bool;
         resB : Byte;
         Niv_SPR : Int;   // Stärke Spritzen
         Zeit_SPR : Int;   // Zeit Spritzen
         Niv_Luft : Int;   // Stärke Lufteinblasung
         Zeit_Luft : Int;   // Zeit Lufteinblasung
         Niv_NS : Int;   // Niveau Füllstand in %
         Zeit_NS : Int;   // Nachspeisezeit getaktete NS
         NS_Kor_Tr : Byte;   // Korrektur Nachspeisezeit für Trommel
         Coun_Kor : Byte;   // Counter Korrektur Nachspeisung
         resD : DInt;
         resR_1 : Real;
         resR_2 : Real;
         resR_3 : Real;
         resI_1 : Int;
         resI_2 : Int;
         ExpoTol : DInt;   // Toleranz Expozeit
         SonDW1 : DInt;   // freie Nutzung Gesamtzeit Rüttler
         SonDW2 : DInt;   // freie Nutzung Intervall ein Rüttler
         SonDW3 : DInt;   // freie Nutzung Intervall aus Rüttler
         SonDW4 : DInt;   // freie Nutzung (Verzögerung US-Rüttler)
         T_Zt_SR : Int;   // Test-Zeit Spritzregister
         T_Zt_NS : Int;   // Test-Zeit Nachspeisung
      END_STRUCT;
   END_VAR
BEGIN
   Pos[1..9].Prio_Pos := 16#05;
   Pos[10].Prio_Pos := 16#00;
   Pos[11..12].Prio_Pos := 16#01;
   Pos[13..14].Prio_Pos := 16#00;
   Pos[15..16].Prio_Pos := 16#01;
   Pos[17].Prio_Pos := 16#00;
   Pos[18].Prio_Pos := 16#01;
   Pos[19].Prio_Pos := 16#00;
   Pos[20..21].Prio_Pos := 16#01;
   Pos[22].Prio_Pos := 16#00;
   Pos[23].Prio_Pos := 16#02;
   Pos[24..27].Prio_Pos := 16#05;
   Pos[28].Prio_Pos := 16#02;
   Pos[29].Prio_Pos := 16#03;
   Pos[30].Prio_Pos := 16#02;
   Pos[1..30].lngsm_IN := FALSE;
   Pos[1..30].lngsm_OUT := FALSE;
   Pos[1..30].res := FALSE;
   Pos[1..30].res1 := FALSE;
   Pos[1..30].res2 := FALSE;
   Pos[1..30].res3 := FALSE;
   Pos[1..30].Luft_Ein := FALSE;
   Pos[1..30].Luft_Auto := FALSE;
   Pos[1].Verweilzeit := 0;
   Pos[2].Verweilzeit := 2107;
   Pos[3].Verweilzeit := 2074;
   Pos[4].Verweilzeit := 0;
   Pos[5].Verweilzeit := 32100;
   Pos[6..7].Verweilzeit := 0;
   Pos[8].Verweilzeit := 115;
   Pos[9..23].Verweilzeit := 0;
   Pos[24].Verweilzeit := 300;
   Pos[25..27].Verweilzeit := 0;
   Pos[28].Verweilzeit := 32;
   Pos[29].Verweilzeit := 1;
   Pos[30].Verweilzeit := 0;
   Pos[1..30].KF_A := 1000.0;
   Pos[1..30].KF_Expo := 1.0;
   Pos[1..30].T_Vorruf := 0;
   Pos[1..30].T_Pend := 1;
   Pos[1..2].T_ATZ := 0;
   Pos[3..7].T_ATZ := 10;
   Pos[8..9].T_ATZ := 5;
   Pos[10].T_ATZ := 10;
   Pos[11..12].T_ATZ := 5;
   Pos[13..14].T_ATZ := 10;
   Pos[15..16].T_ATZ := 5;
   Pos[17].T_ATZ := 10;
   Pos[18].T_ATZ := 5;
   Pos[19].T_ATZ := 10;
   Pos[20..21].T_ATZ := 5;
   Pos[22].T_ATZ := 10;
   Pos[23].T_ATZ := 5;
   Pos[24..27].T_ATZ := 2;
   Pos[28].T_ATZ := 0;
   Pos[29].T_ATZ := 5;
   Pos[30].T_ATZ := 2;
   Pos[1..30].NS_Auto := FALSE;
   Pos[1..25].SR_Auto := FALSE;
   Pos[26].SR_Auto := TRUE;
   Pos[27..29].SR_Auto := FALSE;
   Pos[30].SR_Auto := TRUE;
   Pos[1..30].res6 := FALSE;
   Pos[1..30].WBE_Ein := FALSE;
   Pos[1..30].WBE_Auto := FALSE;
   Pos[1..30].TS_Pos := FALSE;
   Pos[1..30].res9 := FALSE;
   Pos[1..30].res10 := FALSE;
   Pos[1..30].resB := 16#00;
   Pos[1..30].Niv_SPR := 0;
   Pos[1..30].Zeit_SPR := 0;
   Pos[1..30].Niv_Luft := 0;
   Pos[1..30].Zeit_Luft := 0;
   Pos[1..30].Niv_NS := 0;
   Pos[1..30].Zeit_NS := 0;
   Pos[1..30].NS_Kor_Tr := 16#00;
   Pos[1..30].Coun_Kor := 16#00;
   Pos[1..30].resD := 0;
   Pos[1..30].resR_1 := 0.0;
   Pos[1..30].resR_2 := 0.0;
   Pos[1..30].resR_3 := 0.0;
   Pos[1..30].resI_1 := 0;
   Pos[1..30].resI_2 := 0;
   Pos[1..9].ExpoTol := 600;
   Pos[10..22].ExpoTol := 0;
   Pos[23..27].ExpoTol := 600;
   Pos[28..30].ExpoTol := 60;
   Pos[1..30].SonDW1 := 0;
   Pos[1..30].SonDW2 := 0;
   Pos[1..30].SonDW3 := 0;
   Pos[1..30].SonDW4 := 0;
   Pos[1..30].T_Zt_SR := 0;
   Pos[1..30].T_Zt_NS := 0;
END_DATA_BLOCK

DATA_BLOCK "DB_Sperrbereiche"   // DB68
{ S7_Optimized_Access := 'FALSE' }
// stored: AutoNumber false
   VAR RETAIN
      Anzahl : Int := 4;   // * Anzahl der definierten Sperrbereiche
      resD : DInt := 0;
      resw : Int := 0;
      DG1_aktiv : Bool := FALSE;
      DG1_Quit : Bool := FALSE;
      DG1_FP_Taste : Bool := FALSE;
      DG1_Req : Bool := FALSE;
      DG2_aktiv : Bool := FALSE;
      DG2_Quit : Bool := FALSE;
      DG2_FP_Taste : Bool := FALSE;
      DG2_Req : Bool := FALSE;
      Sperre_links : Bool := FALSE;
      Sperre_rechts : Bool := FALSE;
      res3 : Bool := FALSE;
      res4 : Bool := FALSE;
      res5 : Bool := FALSE;
      res6 : Bool := FALSE;
      res7 : Bool := FALSE;
      res8 : Bool := FALSE;
      Bereich : Array[1..5] of Struct   // * Feldlänge anpassen
         aktiv : Bool;   // Bereich ist gesperrt
         min_Inc : DInt;   // untere Grenze Sperrbereich
         max_Inc : DInt;   // obere Grenze Sperrbereich
      END_STRUCT;
   END_VAR
BEGIN
   Bereich[1..5].aktiv := FALSE;
   Bereich[1].min_Inc := 1242;
   Bereich[2].min_Inc := 4938;
   Bereich[3].min_Inc := 1242;
   Bereich[4].min_Inc := 4130;
   Bereich[5].min_Inc := 0;
   Bereich[1].max_Inc := 3372;
   Bereich[2].max_Inc := 7901;
   Bereich[3].max_Inc := 4100;
   Bereich[4].max_Inc := 8654;
   Bereich[5].max_Inc := 0;
END_DATA_BLOCK

DATA_BLOCK "DB_Variantenbefehl"   // DB43
{ S7_Optimized_Access := 'FALSE' }
// stored: AutoNumber false
   VAR RETAIN
      Anzahl_Varianten : Int := 1;   // vorläufige Platzhaltervariable
      Offset : Int := 10;   // Beginn der Daten
      max_Var : Int := 6;   // maximale Anzahl von Varianten (ENTSPRICHT DER FELDLÄNGE)
      resW : Int := 0;
      resW1 : Int := 0;
      Variante : Array[0..1] of Struct
         Pos : Array[1..6] of Byte;
      END_STRUCT;
   END_VAR
BEGIN
   Variante[0].Pos[1] := 16#16;
   Variante[0].Pos[2] := 16#13;
   Variante[0].Pos[3] := 16#11;
   Variante[0].Pos[4] := 16#0E;
   Variante[0].Pos[5] := 16#0D;
   Variante[0].Pos[6] := 16#0A;
   Variante[1].Pos[1..6] := 16#00;
END_DATA_BLOCK

DATA_BLOCK "DB_Zwangsziel"   // DB67
{ S7_Optimized_Access := 'FALSE' }
// stored: AutoNumber false
   VAR RETAIN
      Ziel_von_Pos : Array[0..30] of Byte;   // * Feldlänge anpassen
   END_VAR
BEGIN
END_DATA_BLOCK

DATA_BLOCK "FU_In_Out"   // DB222
{ S7_Optimized_Access := 'FALSE' }
// stored: AutoNumber false
   VAR RETAIN
      Anzahl : Int := 7;   // * Anzahl der zu bedienenden FUs
      Offset : Int := 10;   // * Beginn Daten erster FU
      Leng : Int := 16;   // * Länge einer FU-Struktur
      Fehler_Quitt : Bool := TRUE;
      res1 : Bool := FALSE;
      res2 : Bool := FALSE;
      res3 : Bool := FALSE;
      res4 : Bool := FALSE;
      res5 : Bool := FALSE;
      res6 : Bool := FALSE;
      res7 : Bool := FALSE;
      resB : Byte := 16#00;
      akt_FU : Int := 0;   // Zähler für FU-Bearbeitung
      FU : Array[1..15] of Struct
         Adresse : Int;   // * Adresse EA
         Fehler : Bool;   // Fehlerstatus Altmerker
         res : Bool;
         res1 : Bool;
         res2 : Bool;
         res3 : Bool;
         res4 : Bool;
         res5 : Bool;
         res6 : Bool;
         AM_Fehlernummer : USInt;   // Altmerker Fehlernummer
         PE : Struct
            Statusbyte : Struct
               Fehlernummer : USInt;   // nur bei Stoerung/Warunung
               Endfrei : Bool;   // Freigabe Endstufe
               Bereit : Bool;   // FU betriebsbereit
               PA_Dat : Bool;   // PA Daten freigegeben
               Akt_Intsatz : Bool;   // aktueller Integratorsatz
               Akt_Parsatz : Bool;   // aktueller Parametersatz
               Stoer : Bool;   // Stoerung/Warnung
               End_rechts : Bool;   // Endschalter rechts aktiv
               End_links : Bool;   // Endschalter links aktiv
            END_STRUCT;
            Speed : Int;
            Reserve : Word;
         END_STRUCT;
         PA : Struct
            Steuerwort : Struct
               resB : Byte;
               RegSp : Bool;   // Reglersperre
               FrgStop : Bool;   // Freigabe/Schnellstop
               FrgHalt : Bool;   // Freigabe/Halt
               HaltRg : Bool;   // Haltregelung
               IntUms : Bool;   // Integrator-Umschaltung
               ParUms : Bool;   // Parametersatz-Umschaltung
               Reset : Bool;   // Reset
               res : Bool;
            END_STRUCT;
            Speed : Int;
            Reserve : Word;
         END_STRUCT;
      END_STRUCT;
   END_VAR
BEGIN
   FU[1].Adresse := 1010;
   FU[2].Adresse := 1020;
   FU[3].Adresse := 1030;
   FU[4].Adresse := 1040;
   FU[5].Adresse := 1050;
   FU[6].Adresse := 1060;
   FU[7].Adresse := 1070;
   FU[8].Adresse := 1080;
   FU[9].Adresse := 1090;
   FU[10].Adresse := 0;
   FU[1..10].Fehler := FALSE;
   FU[1..10].res := FALSE;
   FU[1..10].res1 := FALSE;
   FU[1..10].res2 := FALSE;
   FU[1..10].res3 := FALSE;
   FU[1..10].res4 := FALSE;
   FU[1..10].res5 := FALSE;
   FU[1..10].res6 := FALSE;
   FU[1..10].AM_Fehlernummer := 16#00;
   FU[1..10].PE.Statusbyte.Fehlernummer := 16#00;
   FU[1..10].PE.Statusbyte.Endfrei := FALSE;
   FU[1..10].PE.Statusbyte.Bereit := FALSE;
   FU[1..10].PE.Statusbyte.PA_Dat := FALSE;
   FU[1..10].PE.Statusbyte.Akt_Intsatz := FALSE;
   FU[1..10].PE.Statusbyte.Akt_Parsatz := FALSE;
   FU[1..10].PE.Statusbyte.Stoer := FALSE;
   FU[1..10].PE.Statusbyte.End_rechts := FALSE;
   FU[1..10].PE.Statusbyte.End_links := FALSE;
   FU[1..5].PE.Speed := 0;
   FU[6].PE.Speed := 6750;
   FU[7..10].PE.Speed := 0;
   FU[1..10].PE.Reserve := 16#0000;
   FU[1..10].PA.Steuerwort.resB := 16#00;
   FU[1..4].PA.Steuerwort.RegSp := FALSE;
   FU[5].PA.Steuerwort.RegSp := TRUE;
   FU[6].PA.Steuerwort.RegSp := FALSE;
   FU[7..9].PA.Steuerwort.RegSp := TRUE;
   FU[10].PA.Steuerwort.RegSp := FALSE;
   FU[1..5].PA.Steuerwort.FrgStop := FALSE;
   FU[6].PA.Steuerwort.FrgStop := TRUE;
   FU[7..10].PA.Steuerwort.FrgStop := FALSE;
   FU[1..5].PA.Steuerwort.FrgHalt := FALSE;
   FU[6].PA.Steuerwort.FrgHalt := TRUE;
   FU[7..10].PA.Steuerwort.FrgHalt := FALSE;
   FU[1..10].PA.Steuerwort.HaltRg := FALSE;
   FU[1..10].PA.Steuerwort.IntUms := FALSE;
   FU[1..10].PA.Steuerwort.ParUms := FALSE;
   FU[1..10].PA.Steuerwort.Reset := FALSE;
   FU[1..10].PA.Steuerwort.res := FALSE;
   FU[1..5].PA.Speed := 0;
   FU[6].PA.Speed := 6750;
   FU[7..10].PA.Speed := 0;
   FU[1..10].PA.Reserve := 16#0000;
END_DATA_BLOCK

DATA_BLOCK "DB_PNOZ_Comm"   // DB360
{ S7_Optimized_Access := 'FALSE' }
// stored: AutoNumber false
   VAR
      Global_Status : Int;   // 0: OFF; 1: CONNECT; 2: WRITE; 3: READ; 4: DISCONNECT; 5: ERROR
      connection : Struct
         activate : Bool := TRUE;
         established : Bool;   // E
      END_STRUCT;
      CONNECT : Struct
         Request : Bool := TRUE;
         Done : Bool;
         Busy : Bool;
         Error : Bool;
         ID : Word := WORD#16#0002;
         Status : Word;
      END_STRUCT;
      SEND : Struct
         Request : Bool;
         Done : Bool;
         Busy : Bool;
         Error : Bool;
         ID : Word := WORD#16#0002;
         Status : Word;
         Length : UDInt := 43;
      END_STRUCT;
      RECEIVE : Struct
         EN_R : Bool := TRUE;
         ADHOC : Bool := FALSE;
         NDR : Bool := TRUE;
         Busy : Bool;
         Error : Bool;
         ID : Word := WORD#16#0002;
         Status : Word;
         Length : UDInt := 43;
         Receive_Length : UDInt := 43;
      END_STRUCT;
      DISCONNECT : Struct
         Request : Bool;
         Done : Bool;
         Busy : Bool;
         Error : Bool;
         ID : Word;
         Status : Word;
      END_STRUCT;
      Connection_Param { S7_SetPoint := 'True'} : "PNOZ Comm";
   END_VAR
BEGIN
   Connection_Param.local_device_id := BYTE#16#02;
   Connection_Param.rem_staddr[1] := BYTE#16#0A;
   Connection_Param.rem_staddr[2] := BYTE#16#94;
   Connection_Param.rem_staddr[3] := B#16#22;
   Connection_Param.rem_staddr[4] := BYTE#16#46;
END_DATA_BLOCK

DATA_BLOCK "DB_PNOZ_IN_Out"   // DB361
TITLE = DB99 V0.4
{ S7_Optimized_Access := 'FALSE' }
AUTHOR : MW_CSTS
FAMILY : PNOZmc_p
VERSION : 0.4
// für PNOZmulti m1p ab V5.6
// stored: AutoNumber false
   VAR
      In : Struct
         Header : Array[0..7] of Byte;
         PNOZ_OK : Bool := false;   // kein NotHalt global aktiv
         "NH-T_SS_ok" : Bool;   // NH-Taster Schaltschrank o.k.
         "NH-T_Filter_ok" : Bool;   // NH-Taster Filterstation o.k.
         "NH-T_Vers_ok" : Bool;   // NH-Taster Versorgung o.k.
         "NH-T_Ents_ok" : Bool;   // NH-Taster Entsorgung o.k.
         "NH-T_Vent_ok" : Bool;   // NH-Taster Ventilator o.k.
         NH_Koppl_ok : Bool;   // NH Koppl. Res. o.k.
         NH_MP_ok : Bool;   // NH Mobile Panel o.k.
         Tuer_VS_ok : Bool := false;   // Tür Vorderseite o.k.
         Tuer_RS_ok : Bool;   // Tür Rückseite o.k.
         "SRM_Zu_BG-QM43" : Bool;   // SRM ZU UV GP02.BG-QM43
         "SRM_Auf_BG-QM43" : Bool;   // SRM AUF UV GP02.BG-QM43
         "SRM_Zu_BG-QM44" : Bool;   // SRM ZU UV GP02.BG-QM44
         "SRM_Auf_BG-QM44" : Bool;   // SRM AUF UV GP02.BG-QM44
         Abluft_ok : Bool;   // Abluft o.k.
         Tuer_zu_Seite_GP01 : Bool := false;   // Tür geschlossen Seite GP01
         Tuer_zu_vorn_GP01 : Bool := false;   // Tür geschlossen vorn GP01
         Tuer_zu_vorn_GP02 : Bool := false;   // Tür geschlossen vorn GP02
         FG_zu_HQ01 : Bool := false;   // Filtereinhausung geschloosen HQ01.BG06
         FG_zu_HQ02 : Bool := false;   // Filtereinhausung geschloosen HQ02.BG09
         T_Aktion_MP : Bool := false;   // Aktionstaster MobilePanel
         NH_Frg_TW_QF : Bool := false;   // Freigabe Nothalt Transportsystem
         NH_Frg_Pumpen : Bool := false;   // Freigabe Nothalt Pumpen
         NH_Frg_FP_CM01 : Bool := false;   // Freigabe Nothalt Filterpumpe CM01
         NH_Frg_FP_CM02 : Bool := false;   // Freigabe Nothalt Filterpumpe CM02
         NH_Frg_Deckel : Bool := false;   // Freigabe Not-Halt Deckel
         NH_Frg_RT : Bool := false;   // Freigabe Not-Halt Rolltor
         "res11.3" : Bool;
         "res11.4" : Bool;
         "res11.5" : Bool;
         "res11.6" : Bool;
         "res11.7" : Bool;
         VirtualInput : Array[32..127] of Bool;
         LED_0_Fault : Bool;   // LED 0 Fault
         LED_1_Fault : Bool;   // LED 1 Fault
         LED_Fault : Bool;   // LED Fault
         LED_Diag : Bool;   // LED Diag
         LED_Run_ST : Bool := false;   // LED Run ST
         reserved1 : Bool;   // reserved
         LED_Run_FS : Bool := false;   // LED Run FS
         Data_cons_check_bit : Bool;   // Data consistence check bit
         Table_Nr : Byte;   // Table Nr
         Segment : Struct
            Nr : Byte;
            Byte_0 : Byte;
            Byte_1 : Byte;
            Byte_2 : Byte;
            Byte_3 : Byte;
            Byte_4 : Byte;
            Byte_5 : Byte;
            Byte_6 : Byte;
            Byte_7 : Byte;
            Byte_8 : Byte;
            Byte_9 : Byte;
            Byte_10 : Byte;
            Byte_11 : Byte;
            Byte_12 : Byte;
         END_STRUCT;
         reserviert : Byte;
         Checksum : Byte := BYTE#16#0;   // Checksumme, Byte 4 + Byte 39
         Endekennung : Byte := BYTE#16#10;   // last Byte, must be 0x10 every time!
         Struct_Auffueller : Byte;
      END_STRUCT;
      Out : Struct
         Header : Array[0..7] of Byte;
         T_NH_Quitt : Bool;   // Taster Not-Halt Quittierung
         Frg_Automatik : Bool;   // Freigabe Automatik Transportsystem
         res_2 : Bool;
         res_3 : Bool;
         res_4 : Bool;
         res_5 : Bool;
         res_6 : Bool;
         res_7 : Bool;
         res_8 : Bool;
         res_9 : Bool;
         res_10 : Bool;
         res_11 : Bool;
         res_12 : Bool;
         res_13 : Bool;
         res_14 : Bool;
         res_15 : Bool;
         VirtualOutput : Array[16..127] of Bool;
         LED : Byte;
         Req_Table_Nr : Byte;   // Table Nr
         Segment : Struct
            Req_Nr : Byte;
            Byte_0 : Byte;
            Byte_1 : Byte;
            Byte_2 : Byte;
            Byte_3 : Byte;
            Byte_4 : Byte;
            Byte_5 : Byte;
            Byte_6 : Byte;
            Byte_7 : Byte;
            Byte_8 : Byte;
            Byte_9 : Byte;
            Byte_10 : Byte;
            Byte_11 : Byte;
            Byte_12 : Byte;
         END_STRUCT;
         reserviert : Byte;
         Checksum : Byte := BYTE#16#A4;   // Checksumme, Byte 4 + Byte 39
         Endekennung : Byte := BYTE#16#10;   // last Byte, must be 0x10 every time!
         Struct_Auffueller : Byte;
      END_STRUCT;
   END_VAR
BEGIN
   In.Header[0] := BYTE#16#05;
   In.Header[1] := BYTE#16#15;
   In.Header[3] := BYTE#16#26;
   In.Header[4] := BYTE#16#DC;
   Out.Header[0] := BYTE#16#05;
   Out.Header[1] := BYTE#16#15;
   Out.Header[3] := BYTE#16#26;
   Out.Header[4] := BYTE#16#5C;
END_DATA_BLOCK

DATA_BLOCK "DB_PNOZ_Receive"   // DB364
{ S7_Optimized_Access := 'FALSE' }
// stored: AutoNumber false
   VAR
      In : Struct
         Header : Array[0..7] of Byte;
         VirtualInput : Array[0..127] of Bool;
         LED_0_Fault : Bool;   // LED 0 Fault
         LED_1_Fault : Bool;   // LED 1 Fault
         LED_Fault : Bool;   // LED Fault
         LED_Diag : Bool;   // LED Diag
         LED_Run_ST : Bool := false;   // LED Run
         reserved1 : Bool;   // reserved
         LED_Run_FS : Bool := false;   // reserved
         Data_cons_check_bit : Bool;   // Data consistence check bit
         Table_Nr : Byte;   // Table Nr
         Segment : Struct
            Nr : Byte;
            Byte_0 : Byte;
            Byte_1 : Byte;
            Byte_2 : Byte;
            Byte_3 : Byte;
            Byte_4 : Byte;
            Byte_5 : Byte;
            Byte_6 : Byte;
            Byte_7 : Byte;
            Byte_8 : Byte;
            Byte_9 : Byte;
            Byte_10 : Byte;
            Byte_11 : Byte;
            Byte_12 : Byte;
         END_STRUCT;
         reserviert : Byte;
         Checksum : Byte := BYTE#16#0;   // Checksumme, Byte 4 + Byte 39
         Endekennung : Byte := BYTE#16#10;   // last Byte, must be 0x10 every time!
      END_STRUCT;
   END_VAR
BEGIN
   In.Header[0] := BYTE#16#05;
   In.Header[1] := BYTE#16#15;
   In.Header[3] := BYTE#16#26;
   In.Header[4] := BYTE#16#DC;
   In.VirtualInput[0] := TRUE;
   In.VirtualInput[18..23] := TRUE;
   In.VirtualInput[35..36] := TRUE;
END_DATA_BLOCK

DATA_BLOCK "DB_PNOZ_Send"   // DB363
{ S7_Optimized_Access := 'FALSE' }
// stored: AutoNumber false
   VAR
      Out : Struct
         Header : Array[0..7] of Byte;
         VirtualOutput : Array[0..127] of Bool;
         LED : Byte;
         Req_Table_Nr : Byte;   // Table Nr
         Segment : Struct
            Req_Nr : Byte;
            Byte_0 : Byte;
            Byte_1 : Byte;
            Byte_2 : Byte;
            Byte_3 : Byte;
            Byte_4 : Byte;
            Byte_5 : Byte;
            Byte_6 : Byte;
            Byte_7 : Byte;
            Byte_8 : Byte;
            Byte_9 : Byte;
            Byte_10 : Byte;
            Byte_11 : Byte;
            Byte_12 : Byte;
         END_STRUCT;
         reserviert : Byte;
         Checksum : Byte := BYTE#16#A4;   // Checksumme, Byte 4 + Byte 39
         Endekennung : Byte := BYTE#16#10;   // last Byte, must be 0x10 every time!
         Struct_Auffueller : Byte;
      END_STRUCT;
   END_VAR
BEGIN
   Out.Header[0] := BYTE#16#05;
   Out.Header[1] := BYTE#16#15;
   Out.Header[3] := BYTE#16#26;
   Out.Header[4] := BYTE#16#5C;
END_DATA_BLOCK

